// TIA Portal V20 program export: 1 tag tables, 54 data types, 39 data blocks, 33 code blocks (in call order from the OBs), 10 instance data blocks

VAR_GLOBAL   // PLC tag table "默认变量表"
   Clock_Byte AT %MB0 : Byte;
   Clock_10Hz AT %M0.0 : Bool;
   Clock_5Hz AT %M0.1 : Bool;
   "Clock_2.5Hz" AT %M0.2 : Bool;
   Clock_2Hz AT %M0.3 : Bool;
   "Clock_1.25Hz" AT %M0.4 : Bool;
   Clock_1Hz AT %M0.5 : Bool;
   "Clock_0.625Hz" AT %M0.6 : Bool;
   "Clock_0.5Hz" AT %M0.7 : Bool;
   System_Byte AT %MB1 : Byte;
   FirstScan AT %M1.0 : Bool;
   DiagStatusUpdate AT %M1.1 : Bool;
   AlwaysTRUE AT %M1.2 : Bool;
   AlwaysFALSE AT %M1.3 : Bool;
   PositioningAxis_1_Actor_Interface_AddressIn AT %I129.0 : "PD_TEL5_IN";
   PositioningAxis_1_Actor_Interface_AddressOut AT %Q132.0 : "PD_TEL5_OUT";
   滑台伺服S200_Actor_Interface_AddressIn AT %I260.0 : "PD_TEL105_IN";
   滑台伺服S200_Actor_Interface_AddressOut AT %Q260.0 : "PD_TEL105_OUT";
   RLO_1 AT %M100.0 : Bool;
   RLO_0 AT %M100.1 : Bool;
   FirstCycle AT %M100.2 : Bool;
   S120正限位 AT %I0.0 : Bool;
   s120负限位 AT %I0.1 : Bool;
   s120原点信号 AT %I0.2 : Bool;
   滑台伺服S200_Actor_Interface_TorqueDataAddressIn AT %I280.0 : "PD_TEL750_IN";
   滑台伺服S200_Actor_Interface_TorqueDataAddressOut AT %Q280.0 : "PD_TEL750_OUT";
   S200原点信号 AT %I0.3 : Bool;
   S200正限位 AT %I0.4 : Bool;
   S200负限位 AT %I0.5 : Bool;
   Tag_1 AT %M10.5 : Bool;
   Tag_2 AT %M10.6 : Bool;
END_VAR
VAR_GLOBAL CONSTANT   // user constants
   PN_DevDiag_MaxModules_UserConst : Int := 128;   // Maximale Anzahl der Module in einer ET-Station (z.B. ET200...); WICHTIG: um Zykluszeit und Speicherplatz zu optimieren mögl. kleinen Wert hier einstellen / Max number of modules, for optimization of scantime and memory space keep small / Max 数量 of modules, 给 optimization of scantime 和 内存 space keep small
   PN_DevDiag_MaxDevices_UserConst : Int := 255;   // Maximale Anzahl der PN-Devices; WICHTIG: um Zykluszeit und Speicherplatz zu optimieren mögl. kleinen Wert hier einstellen / Max number of PN-devices, for optimization of scantime and memory space keep small / Max 数量 of PN-devices, 给 optimization of scantime 和 内存 space keep small
   Type_HMI : Int := 101;   // SICAR HMI / HMI
   "Type_HMI+External" : Int := 102;   // SICAR HMI&Ext. / HMI&External / SICAR HMI&外部
   Type_External : Int := 103;   // SICAR Ext / External / SICAR 外部
   Type_OperatorPanel : Int := 105;   // SICAR OperatorPanel / OperatorPanel
   No_of_DataSets_Counter : Int := 8;   // Anzahl Datensätze Zähler / Number of data sets Counter / 数量 of 数据 sets 计数器
   No_of_DataSets_ShiftCounter : Int := 8;   // Anzahl Datensätze Schichtzähler / Number of data sets Shift Counter / 数量 of 数据 sets 工作轮班 计数器
   No_of_DataSets_CycleTimer : Int := 8;   // Anzahl Datensätze Taktzeiten / Number of data sets Cycle Timer / 数量 of 数据 sets 周期 记时器
   No_of_DataSets_LimitValues : Int := 8;   // Anzahl Datensätze Grenzwerte / Number of data sets Limit Value / 数量 of 数据 sets 限制 值
   No_Drives : Int := 2;   // Anzahl Antriebe / Number of drives / 数量 of 驱动
   No_UserOperation_screens : Int := 2;   // Anzahl Anwender Bedien-Bilder / Number of UserOperation screens / 数量 of UserOperation screens
   No_OperationMODE : Int := 5;   // Anzahl verwendeter Betriebsarten Breiche (max.: 12) / Number of used operation mode areas (max.: 12 ) / 数量 of used 运行 模式 areas (max.: 12 )
   No_HMI_PANEL : Int := 5;   // Anzahl verwendeter HMI/Panel (Max.: 40: 8 HMIs + 32 Panels) / Number of used HMI/Panel (Max.: 40: 8 HMIs + 32 Panels) / 数量 of used HMI/Panel (Max.: 40: 8 HMIs + 32 Panels)
   EQUIPMENTDATA_STEPHISTORYLENGTH : Int := 149;   // Equipment Data Step History Array Length / 设备 数据 步 历史 Array 长度
   EQUIPMENTDATA_ACTIVEALARMSLENGTH : Int := 9;   // Equipment Data Active Alarms Array Length / 设备 数据 现行 警报 Array 长度
   No_Reader : Int := 5;   // Anzahl Lesestellen / Number of reader / 数量 of 读码器
   No_Fixtures : Int := 2;
   No_Valves : Int := 4;
   No_PP : Int := 4;
   OpMode07_No_Robot : Int := 4;   // Anzahl Antriebe / Number of Robots
   No_ES : Int := 4;   // Anzahl Antriebe / Number of drives
   No_GS : Int := 1;   // Anzahl Antriebe / Number of drives
   No_LC : Int := 1;   // Anzahl Antriebe / Number of drives
   No_LS : Int := 1;   // Anzahl Antriebe / Number of drives
   Single_Input : Int := 1;
   OSSD_Input : Int := 5;
   OP_Sum : SInt := 2;   // 工位总数
   HMI_AXISCTRL_COUNT_AXES_UPPER_LIM : Int := 5;   // Upper limit for number of axes in HMI (maximum number - 1)
END_VAR

TYPE "ConvHMICMD"
   STRUCT
      StationOnly : Bool;   // Run Within Station Only
      SafetyTest : Bool;   // Safety Test
      Spare1 : Bool;   // Spare
      Spare2 : Bool;   // Spare
      Spare3 : Bool;   // Spare
      Spare4 : Bool;   // Spare
      Spare5 : Bool;   // Spare
      Spare6 : Bool;   // Spare
      Spare7 : Bool;   // Spare
      Spare8 : Bool;   // Spare
      Spare9 : Bool;   // Spare
      Spare10 : Bool;   // Spare
      Spare11 : Bool;   // Spare
      Spare12 : Bool;   // Spare
      Spare13 : Bool;   // Spare
      Spare14 : Bool;   // Spare
      Spare15 : Bool;   // Spare
      Spare16 : Bool;   // Spare
      Spare17 : Bool;   // Spare
      Spare18 : Bool;   // Spare
      Spare19 : Bool;   // Spare
      Spare20 : Bool;   // Spare
      Spare21 : Bool;   // Spare
      Spare22 : Bool;   // Spare
      Spare23 : Bool;   // Spare
      Spare24 : Bool;   // Spare
      Spare25 : Bool;   // Spare
      Spare26 : Bool;   // Spare
      Spare27 : Bool;   // Spare
      Spare28 : Bool;   // Spare
      Spare29 : Bool;   // Spare
      Spare30 : Bool;   // Spare
   END_STRUCT;
END_TYPE

TYPE "InPut"
   STRUCT
      TrfInSetBegin : Bool;   // Command in from Graph / Load Begin: condition to start transfer IN set
      TrfInSetIntlkOk : Bool;   // Transfer IN Interlock Set OK
      TrfInResIntlkOk : Bool;   // Transfer IN Interlock Reset OKt
      TrfOutSetBegin : Bool;   // Unload Begin: condition to start transfer OUT set
      TrfOutSetIntlkOk : Bool;   // Transfer Out Interlock Set Ok
      TrfOutResIntlkOk : Bool;   // Transfer OUT Interlock Reset Ok
      TrfOutResBegin : Bool;
   END_STRUCT;
END_TYPE

TYPE "OutPut"
   STRUCT
      Active : Bool;   // Roller is Active
      TrfInSetRdyRcv : Bool;   // Ready to Receive: Signal to previous object set
      TrfInSetArrived : Bool;   // Body Arrived: Signal to previous object Set
      TrfInSetActive : Bool;   // Transfer in set active
      TrfInSetFinished : Bool;   // Transfer in set finished
      TrfOutSetRdyDlv : Bool;   // Ready to Deliver: Signal to next object set
      TrfOutSetTM : Bool;   // Transfer: Signal to next object set
      TrfOutSetActive : Bool;   // Transfer out set active
      TrfOutSetFinished : Bool;   // Transfer out set finished
      TrfInResRdyRcv : Bool;   // Ready to Receive: Signal to previous object Reset
      TrfInResArrived : Bool;   // Body Arrived: Signal to previous object Reset
      TrfInResActive : Bool;   // Transfer in Reset active
      TrfInResFinished : Bool;   // Transfer in Reset finished
      TrfOutResRdyDlv : Bool;   // Ready to Deliver: Signal to next object Reset
      TrfOutResTM : Bool;   // Transfer: Signal to next object Reset
      TrfOutResActive : Bool;   // Transfer out Reset active
      TrfOutResFinished : Bool;   // Transfer out Reset finished
      BodyInPosition : Bool;   // Body In Position / Body in Position on roller
      NoSkid : Bool;   // No Skid
      LSpdSet : Bool;   // Lower Speed Set
      HSpdSet : Bool;   // Hight Speed Set
      SelectLower : Bool;   // Selext Lower Speed
   END_STRUCT;
END_TYPE

TYPE "RollBed"
   STRUCT
      HMI : "H_HMI";
      G120 { S7_SetPoint := 'True'} : "H_Roller2W2S-G120PN";
      Config { S7_SetPoint := 'True'} : "RollerConvConfig";
      InPut : "InPut";
      OutPut : "OutPut";
   END_STRUCT;
END_TYPE

TYPE "RollerConvConfig"
   STRUCT
      DeadEnd : Bool;   // Dead End Disable Positiong Fault
      TrspNoLowSpeed : Bool;   // Input 14
      StopDetSetUsed : Bool;   // Input 0
      LowSpeedDetSetUsed : Bool;   // Low Speed Det Used
      LowSpeedDetSetConstOn : Bool;   // Low Speed Sensor Constant on
      StopDetResUsed : Bool;   // Stop detection Reset used
      LowSpeedDetResUsed : Bool;   // Input 10
      LowSpeedDetResConstOn : Bool;   // Lowspeed stop detection Constant On
      TrainActivatedSet : Bool;   // Train transport used set direction
      TrfInSetUsed : Bool;   // Transfer In Set Used
      TrfOutSetUsed : Bool;   // Transfer Out Reset Used
      TrainActivatedRes : Bool;   // Train transport used Reset direction
      TrfInResUsed : Bool;   // Transfer In Reset Used
      TrfOutResUsed : Bool;   // Transfer Out Reset Used
      EnableAlarmHW : Bool := TRUE;   // Enable Alarm hardware (e.g. Safetyswitch, Motorprotector, detections)
      EnableAlarmTransfer : Bool;   // Enable Alarm transfer (e.g. Transfer in , transfer out)
      EnableG120Reset : Bool;   // Enable Driver Reset
      EnableCheckSpeedOK : Bool;   // Enable Speed checking on the G120 Driver
      EnableSetpoint : Bool;   // Enable setpoint
      EnableRFG : Bool;   // Follow setpoint
      NotQuickStop : Bool;   // QuickStop function; When FALSE the QuickStop of the G120 is Active
      NotImmediateStop : Bool;   // Immediate function; When FALSE the immediate stop of the G120 is Active
      EnableBeltControlSetDet : Bool;   // Config Belt Control
      EnableBeltControlResDet : Bool;   // Config Belt Control
      SLSUsed : Bool;   // Profisafe SLS Configuration Used
      SafetySwUsed : Bool;   // Input 12
      SafetySwNc : Bool;   // Input 15
      ReleaseBrakeUsed : Bool;   // Input 13
      RearDetUsed : Bool;   // Input 9
      RevSwUsed : Bool;   // Input 8
      MotorProtectionUsed : Bool;   // Motorprotection Used
      MotorProtectionNc : Bool;   // Motorprotection NC
      InitDirection : Bool;   // Input 6
      ForceManual : Bool;   // Configuration
      Spare1 : Bool;   // Spare
      Spare2 : Bool;   // Spare
      Spare3 : Bool;   // Spare
      TrfMaxTime : DInt;   // Max allowed transfertime (millisec)
      RPMSpeed : Real;   // Movment Rpm
      EnableRPMSpeed : Bool;   // Enable RPM Speed
      ReferenceSpeed : Int;   // Reference value for speed, stored in P2000 ot the SINAMICS
      ReferenceCurrent : Real;   // Reference value for current, stored in P2002 ot the SINAMICS
      ReferenceTorque : Real;   // Reference value for torque, stored in P2003 ot the SINAMICS
      DelaySetStopDet : Time := T#1ms;   // Delay Time Stop Detection
      DelayResStopDet : Time := T#1ms;   // Delay Time Stop Detection
      HWSubInput : HW_SUBMODULE;   // Address (input/output)
      HWSubOutput : HW_SUBMODULE;   // I/O
      SafetyAddress : HW_SUBMODULE;   // Address (input/output)
      FilterBeltControlSec : DInt;   // Filter In Seconds Belt Control
   END_STRUCT;
END_TYPE

TYPE "Rollerbed_Configuration"
   STRUCT
      StopDetSetUsed : Bool;
      LowSpeedDetSetUsed : Bool;
      LSpeedDetSetConstOn : Bool;
      TrainActivatedSet : Bool;
      TrfInSetUsed : Bool;
      TrfOutSetUsed : Bool;
      TrspNoLowSpeed : Bool;
      InitDirection : Bool;
      RevSwUsed : Bool;
      StopDetResUsed : Bool;
      LowSpeedDetResUsed : Bool;
      LSpeedDetResConstOn : Bool;
      TrainActivatedRes : Bool;
      TrfInResUsed : Bool;
      TrfOutResUsed : Bool;
      SafetySwNc : Bool;
      SafetySwUsed : Bool;
      ReleaseBrakeUsed : Bool;
      MotorProtectionSwNc : Bool;
      MotorProtectionUsed : Bool;
   END_STRUCT;
END_TYPE

TYPE "sPos16"
   STRUCT
      I_SS_bHome : Bool;   // 原点传感器
      I_SS_bFW : Bool := TRUE;   // 前限位
      I_SS_bBW : Bool := TRUE;   // 后限位
      I_CMD_bEnableAxis : Bool;   // 使能
      I_CMD_bResetAxis : Bool;   // 复位
      I_CMD_bjogForward : Bool;   // Taster Aufwärts / 正点
      I_CMD_bjogBackward : Bool;   // Taster Abwärts / 反点
      I_CMD_bmoveVelocity : Bool;   // 速度运行
      I_CMD_bstop : Bool;   // 停止
      I_CMD_bfastStop : Bool;   // 急停
      I_CMD_bHoming : Bool;   // 回零
      I_CMD_bGoToPos : Array[0..15] of Bool;   // Start Aufwärts in Automatik / 16个定位
      I_CMD_iGoToPos : Word;   // 16个定位 Word
      I_CMD_bCallAbsPos : Bool;   // 定位位置切换时，单独的定位按钮
      I_CMD_bRelPos : Bool;   // 相对定位
      I_CMD_MyBool : Array[0..5] of Bool;   // 临时变量
      I_Para_rJog_Speed : Array[0..2] of LReal;   // 点动速度/ACC/DEC/JERK
      I_Para_rMV_Speed : Array[0..2] of LReal;   // 速度运行速度/ACC/DEC/JERK
      I_Para_rStop_Dec : Array[0..1] of LReal;   // 速度运行速度/ACC/DEC/JERK
      I_Para_rEStop_Dec : Array[0..1] of LReal;   // 速度运行速度/ACC/DEC/JERK
      I_Para_iNum_Abspos : Int := 4;
      I_Para_rPos_Abs : Array[0..16] of LReal;   // 绝对定位目标位置
      I_Para_rSpeed_Abs : Array[0..16] of LReal;   // Endlage Unten / 绝对定位速度
      I_Para_rAcc_Set : Array[0..16] of LReal;   // 绝对定位加速度
      I_Para_rDec_Set : Array[0..16] of LReal;   // 绝对定位减速度
      I_Para_rJerk_Set : Array[0..16] of LReal;   // 绝对定位加加速度
      I_Para_rSpeedPercent : LReal := 20.0;   // Endlage Unten / 速度设定百分比
      I_Para_iHomeMode : Int;   // 回零方式
      I_Para_rHomePos : LReal;   // 回零位置
      O_Status_bAxisReady : Bool;   // 轴通讯正常
      O_Status_bAxisEnabled : Bool;   // 轴使能
      O_Status_bjogForward : Bool;   // 轴正点中
      O_Status_bjogBackward : Bool;   // 轴反点中
      O_Status_bHomed : Bool;   // 轴归零完成
      O_Status_bAtHome : Bool;   // 轴在零位
      O_Status_bSstill : Bool;   // 轴静止
      O_Status_bAxisBusy : Bool;   // 轴运行中
      O_Status_bAxisSyned : Bool;   // 同步上
      O_Status_bAxisError : Bool;   // 轴报警
      O_Status_bAtPos : Array[0..15] of Bool;   // Ausgang Aufwärts / 在目标位置上
      O_Status_bPosDone : Array[0..15] of Bool;   // 定位完成
      O_Status_bPosing : Array[0..15] of Bool;   // Ausgang Aufwärts / 定位中
      O_Status_bRelPosDone : Bool;   // 相对定位完成
      O_Status_rActPos : LReal;   // 实际位置
      O_Status_rActSpeed : LReal;   // 实际速度
      O_Status_iAxisFaultNum : UDInt;   // 轴报警代码
      O_Status_iDriveFaultNum : UDInt;   // 驱动报警代码
      O_Status_iFBStatus : Word;   // 运动功能块状态
      O_Status_iMCStatus : Word;   // 运动指令状态
      O_Status_rDriveTorque : LReal;   // 驱动扭矩
      O_Status_rDriveTemp : LReal;   // 驱动温度
      O_Status_rDriveRpm : LReal;   // 驱动转速
      O_Status_AxisName : WString[24] := WSTRING#'No axis';   // Name of axis
      O_Status_mybool : Array[0..5] of Bool;   // 备用
      O_Status_myLreal : Array[0..5] of LReal;   // 备用
      I_InLock_bEnableAxis : Bool;   // 使能
      I_InLock_bResetAxis : Bool;   // 复位
      I_InLock_bjogForward : Bool;   // Taster Aufwärts / 正点
      I_InLock_bjogBackward : Bool;   // Taster Abwärts / 反点
      I_InLock_bmoveVelocity : Bool;   // 速度运行
      I_InLock_bstop : Bool;   // 停止
      I_InLock_bfastStop : Bool;   // 急停
      I_InLock_bHoming : Bool;   // 回零
      I_InLock_bGoToPos : Array[0..16] of Bool;   // Start Aufwärts in Automatik / 16个定位
      I_InLock_iGoToPos : Word;   // 16个定位 Word
      I_InLock_bCallAbsPos : Bool;   // 定位位置切换时，单独的定位按钮
      I_InLock_bRelPos : Bool;   // 相对定位
      I_InLock_MyBool : Array[0..5] of Bool;   // 临时变量
      I_HMI_bEnableAxis : Bool;   // 使能
      I_HMI_bResetAxis : Bool;   // 复位
      I_HMI_bjogForward : Bool;   // Taster Aufwärts / 正点
      I_HMI_bjogBackward : Bool;   // Taster Abwärts / 反点
      I_HMI_bmoveVelocity : Bool;   // 速度运行
      I_HMI_bstop : Bool;   // 停止
      I_HMI_bfastStop : Bool;   // 急停
      I_HMI_bHoming : Bool;   // 回零
      I_HMI_bGoToPos : Array[0..16] of Bool;   // Start Aufwärts in Automatik / 16个定位
      I_HMI_iGoToPos : Word;   // 16个定位 Word
      I_HMI_bCallAbsPos : Bool;   // 定位位置切换时，单独的定位按钮
      I_HMI_bRelPos : Bool;   // 相对定位
      I_HMI_MyBool : Array[0..5] of Bool;   // 临时变量
   END_STRUCT;
   // I_Para_rJog_Speed[0] := 10.0;
   // I_Para_rJog_Speed[1..2] := 30.0;
   // I_Para_rMV_Speed[0] := 20.0;
   // I_Para_rMV_Speed[1..2] := 30.0;
   // I_Para_rStop_Dec[0] := 30.0;
   // I_Para_rStop_Dec[1] := 50.0;
   // I_Para_rEStop_Dec[0..1] := 50.0;
   // I_Para_rPos_Abs[1] := 10.0;
   // I_Para_rPos_Abs[2] := 20.0;
   // I_Para_rPos_Abs[3] := 30.0;
   // I_Para_rPos_Abs[4] := 40.0;
   // I_Para_rPos_Abs[5] := 50.0;
   // I_Para_rPos_Abs[6] := 60.0;
   // I_Para_rPos_Abs[7] := 70.0;
   // I_Para_rPos_Abs[8] := 80.0;
   // I_Para_rPos_Abs[9] := 90.0;
   // I_Para_rPos_Abs[10] := 100.0;
   // I_Para_rPos_Abs[11] := 110.0;
   // I_Para_rPos_Abs[12] := 120.0;
   // I_Para_rPos_Abs[13] := 130.0;
   // I_Para_rPos_Abs[14] := 140.0;
   // I_Para_rPos_Abs[15] := 150.0;
   // I_Para_rPos_Abs[16] := 160.0;
   // I_Para_rSpeed_Abs[0..16] := 20.0;
   // I_Para_rAcc_Set[0..16] := 50.0;
   // I_Para_rDec_Set[0..16] := 50.0;
   // I_Para_rJerk_Set[0..16] := 50.0;
END_TYPE

TYPE "SHIFTMODEL_LIST_UDT"
   STRUCT
      ShiftmodelList_Zero { ExternalAccessible := 'False'; ExternalVisible := 'False'; ExternalWritable := 'False'; S7_SetPoint := 'True'} : "SHIFTMODEL-TIMES_1DAY_UDT";   // Alle Zeitwerte (TOD) gleich 00:00:00 / All Time values (TOD) are 00:00:00
      ShiftmodelList_1 { ExternalAccessible := 'False'; ExternalVisible := 'False'; ExternalWritable := 'False'; S7_SetPoint := 'True'} : "SHIFTMODEL-TIMES_1DAY_UDT";   // Schichtmodel Liste 1 (1 Tag) / Shiftmodel list 1 (1 day)
      ShiftmodelList_2 { ExternalAccessible := 'False'; ExternalVisible := 'False'; ExternalWritable := 'False'; S7_SetPoint := 'True'} : "SHIFTMODEL-TIMES_1DAY_UDT";   // Schichtmodel Liste 2 (1 Tag) / Shiftmodel list 2 (1 day)
      ShiftmodelList_3 { ExternalAccessible := 'False'; ExternalVisible := 'False'; ExternalWritable := 'False'; S7_SetPoint := 'True'} : "SHIFTMODEL-TIMES_1DAY_UDT";   // Schichtmodel Liste 3 (1 Tag) / Shiftmodel list 3 (1 day)
      ShiftmodelList_4 { ExternalAccessible := 'False'; ExternalVisible := 'False'; ExternalWritable := 'False'; S7_SetPoint := 'True'} : "SHIFTMODEL-TIMES_1DAY_UDT";   // Schichtmodel Liste 4 (1 Tag) / Shiftmodel list 4 (1 day)
      ShiftmodelList_5 { ExternalAccessible := 'False'; ExternalVisible := 'False'; ExternalWritable := 'False'; S7_SetPoint := 'True'} : "SHIFTMODEL-TIMES_1DAY_UDT";   // Schichtmodel Liste 5 (1 Tag) / Shiftmodel list 5 (1 day)
      ShiftmodelList_6 { ExternalAccessible := 'False'; ExternalVisible := 'False'; ExternalWritable := 'False'; S7_SetPoint := 'True'} : "SHIFTMODEL-TIMES_1DAY_UDT";   // Schichtmodel Liste 6 (1 Tag) / Shiftmodel list 6 (1 day)
      ShiftmodelList_7 { ExternalAccessible := 'False'; ExternalVisible := 'False'; ExternalWritable := 'False'; S7_SetPoint := 'True'} : "SHIFTMODEL-TIMES_1DAY_UDT";   // Schichtmodel Liste 7 (1 Tag) / Shiftmodel list 7 (1 day)
      ShiftmodelList_8 { ExternalAccessible := 'False'; ExternalVisible := 'False'; ExternalWritable := 'False'; S7_SetPoint := 'True'} : "SHIFTMODEL-TIMES_1DAY_UDT";   // Schichtmodel Liste 8 (1 Tag) / Shiftmodel list 8 (1 day)
      ShiftmodelList_9 { ExternalAccessible := 'False'; ExternalVisible := 'False'; ExternalWritable := 'False'; S7_SetPoint := 'True'} : "SHIFTMODEL-TIMES_1DAY_UDT";   // Schichtmodel Liste 9 (1 Tag) / Shiftmodel list 9 (1 day)
      ShiftmodelList_10 { ExternalAccessible := 'False'; ExternalVisible := 'False'; ExternalWritable := 'False'; S7_SetPoint := 'True'} : "SHIFTMODEL-TIMES_1DAY_UDT";   // Schichtmodel Liste 10 (1 Tag) / Shiftmodel list 10 (1 day)
      Shiftmodel_WeekDay { ExternalAccessible := 'False'; ExternalVisible := 'False'; ExternalWritable := 'False'; S7_SetPoint := 'True'} : Array[1..7] of "SHIFTMODEL-TIMES_1DAY_UDT";   // Schichtmodel 1 Woche (1: Sunday, 2: Monday, 3: Thuesday, 4: Wednesday, 5: Thursday, 6: Friday, 7: Saturday) / Shiftmodel 1 week (1: Sunday, 2: Monday, 3: Thuesday, 4: Wednesday, 5: Thursday, 6: Friday, 7: Saturday)
   END_STRUCT;
END_TYPE

TYPE "RFID_BALLUFF_UDT"
   STRUCT
      Start : Bool;
      job_Type : Int;
      Adr_Recieve : Int;
      Adr_Send : Int;
      Addr_CodeTag : Int;
      Length_CodeTag : Int;
   END_STRUCT;
END_TYPE

TYPE "UDT_RFID_Basic_Data"
   STRUCT
      Pallet_ID : Int;   // 托盘号
      Repair_Status : Int;   // 返修标致（0：无状态，1：正常件，2：返修件）
      Reserves_1 : Int;   // 预留
      Reserves_2 : Int;   // 预留
      Reserves_3 : Int;   // 预留
      Reserves_4 : Int;   // 预留
      Reject_Stn_Number : String[8];   // 拒绝工位（由不合格工位写入）
      UpLoad_Stn_Number : String[8];   // 上线工位（返修上线工位写入）
      Reserves_5 : Int;   // 预留
      PLCProductWorkOrderID : String[66];   // 产品工单号数据
      PLCProductModelID : String[32];   // 产品型号信息
      PLCProductRecipeID : Word;   // 产品配方号数据
      PLCProductSN : String[96];   // 产品序列号
      PLCProductPN : String[96];   // 产品批次号
      PLCCurrentProductSN : String[96];   // 当前处理的产品序列号
      PLCProductCustomerSN : String[96];   // 产品客户序列号
      PLCProductCustomerSNType : Word;   // 产品客户序列号类型
      Reserves_6 : Int;   // 预留
      Reserves_7 : Int;   // 预留
      Reserves_8 : Int;   // 预留
      Reserves_9 : Int;   // 预留
   END_STRUCT;
END_TYPE

TYPE "UDT_RFID_STN_Data"
   STRUCT
      Station_Task : Byte;   // 工位建造状态（0:未完成 1:接受 2:拒绝）
      TASK_01 : Byte;   // 任务1状态（0:未完成 1:接受 2:拒绝）
      TASK_02 : Byte;   // 任务2状态（0:未完成 1:接受 2:拒绝）
      TASK_03 : Byte;   // 任务3状态（0:未完成 1:接受 2:拒绝）
      TASK_04 : Byte;   // 任务4状态（0:未完成 1:接受 2:拒绝）
      TASK_05 : Byte;   // 任务5状态（0:未完成 1:接受 2:拒绝）
      TASK_06 : Byte;   // 任务6状态（0:未完成 1:接受 2:拒绝）
      TASK_07 : Byte;   // 任务7状态（0:未完成 1:接受 2:拒绝）
      TASK_08 : Byte;   // 任务8状态（0:未完成 1:接受 2:拒绝）
      TASK_09 : Byte;   // 任务9状态（0:未完成 1:接受 2:拒绝）
   END_STRUCT;
END_TYPE

TYPE "VAR_RFID_UDT_BALLUFE"
   STRUCT
      Pallte_On { ExternalAccessible := 'False'; ExternalVisible := 'False'; ExternalWritable := 'False'} : Bool;
      Init { ExternalAccessible := 'False'; ExternalVisible := 'False'; ExternalWritable := 'False'} : Bool;   // 初始化
      Read_Req { ExternalAccessible := 'False'; ExternalVisible := 'False'; ExternalWritable := 'False'} : Bool;
      Write_Req { ExternalAccessible := 'False'; ExternalVisible := 'False'; ExternalWritable := 'False'} : Bool;
      Dyn { ExternalAccessible := 'False'; ExternalVisible := 'False'; ExternalWritable := 'False'} : Bool;   // 动态读写
      CT_Type { ExternalAccessible := 'False'; ExternalVisible := 'False'; ExternalWritable := 'False'} : Bool;   // 编码器类型
      IO_Start { ExternalAccessible := 'False'; ExternalVisible := 'False'; ExternalWritable := 'False'} : Int;
      IO_Length { ExternalAccessible := 'False'; ExternalVisible := 'False'; ExternalWritable := 'False'} : Int;
      CT_Length_R { ExternalAccessible := 'False'; ExternalVisible := 'False'; ExternalWritable := 'False'} : Int;
      CT_Length_W { ExternalAccessible := 'False'; ExternalVisible := 'False'; ExternalWritable := 'False'} : Int;
      Send_DB { ExternalAccessible := 'False'; ExternalVisible := 'False'; ExternalWritable := 'False'} : Int;
      Send_Adr { ExternalAccessible := 'False'; ExternalVisible := 'False'; ExternalWritable := 'False'} : Int;
      Recv_DB { ExternalAccessible := 'False'; ExternalVisible := 'False'; ExternalWritable := 'False'} : Int;
      Recv_Adr { ExternalAccessible := 'False'; ExternalVisible := 'False'; ExternalWritable := 'False'} : Int;
      Read_Finished { ExternalAccessible := 'False'; ExternalVisible := 'False'; ExternalWritable := 'False'} : Bool;
      Write_Finished { ExternalAccessible := 'False'; ExternalVisible := 'False'; ExternalWritable := 'False'} : Bool;
      Error { ExternalAccessible := 'False'; ExternalVisible := 'False'; ExternalWritable := 'False'} : Bool;
      ErrorNum { ExternalAccessible := 'False'; ExternalVisible := 'False'; ExternalWritable := 'False'} : Int;
      Dig_In { ExternalAccessible := 'False'; ExternalVisible := 'False'; ExternalWritable := 'False'} : Bool;
      CT_Present { ExternalAccessible := 'False'; ExternalVisible := 'False'; ExternalWritable := 'False'} : Bool;
   END_STRUCT;
END_TYPE

TYPE "MOTOR_LOCK_HMI_UDT"
   STRUCT
      State : DWord;   // Status Tec_Unit / State Tec_unit
      Plant_Identifier : WString[24];   // Betriebsmittel Kennzeichen / Plant identifier
      Move : Word;   // Schnittstelle Bewegungen / Interface Movement/Position
      Position : DWord;   // Schnittstelle Positionen 1-8 / Interface Position
      Alarm : Word;   // Störungen / Alarms
      State_Colour : SInt;   // Status Farbschema / State colour code
      HMI_Control_No : Int;   // HMI-Control Nummer / HMI-Control number
      OPModeArea { ExternalWritable := 'False'} : USInt;   // BA-Bereich / OPMode area
   END_STRUCT;
END_TYPE

TYPE "UDT_FIXTURE_IF"
   STRUCT
      Valves : Array[1..10] of "UDT_VALVE";
      PP : Array[1..35] of "PP_INTERFACE_UDT";
      Process_Complete : Array[1..16] of Bool;
      Work_Pos : Bool;
      Home_Pos : Bool;
      AtKnownPos : Bool;
   END_STRUCT;
END_TYPE

TYPE "UDT_VALVE"
TITLE = DEMO
// Autor: SICAR / Autor: Tesla
   STRUCT
      Auto_Work : Bool;   // Cmd To Move Valve To Work / Cmd 到 移动 汽阀 到 工作位
      Auto_Home : Bool;   // Cmd To Move Valve To Home / Cmd 到 移动 汽阀 到 原位
      At_Work : Bool;   // Status At Work / 状态 在 工作位
      At_Home : Bool;   // Status At Home / 状态 在 原位
      Enable_Work : Bool;   // interlock to move valve to Work / 互锁 到 移动 汽阀 到 工作位
      Enable_Home : Bool;   // interlock to move valve to Home / 互锁 到 移动 汽阀 到 原位
      General_Alarm : Bool;
      Known_Position : Bool;
      Position : "VALVE_POSITION_UDT";   // Feedback from Sensors / 反馈 从 Sensors
   END_STRUCT;
END_TYPE

TYPE "Udt_M200D_IN"
   STRUCT
      "Ready (automatic)" : Bool;
      "Motor on" : Bool;
      "Group fault" : Bool;
      "Group warning" : Bool;
      "Input 1_Stop" : Bool;
      "Input 2_Ocuupy" : Bool;
      "Input 3" : Bool;
      "Input 4" : Bool;
      "Current motor current Icurr % Bit 0" : Bool;
      "Current motor current Icurr % Bit 1" : Bool;
      "Current motor current Icurr % Bit 2" : Bool;
      "Current motor current Icurr % Bit 3" : Bool;
      "Current motor current Icurr % Bit 4" : Bool;
      "Current motor current Icurr % Bit 5" : Bool;
      "Manual mode local mode" : Bool;
      "Ramp operation" : Bool;
   END_STRUCT;
END_TYPE

TYPE "Udt_M200D_OUT"
   STRUCT
      "Motor CW" : Bool;
      "Motor CCW" : Bool;
      "Control for brake" : Bool;
      "Trip reset" : Bool;
      "Emergency start" : Bool;
      "Self-test" : Bool;
      Unassigned1 : Bool;
      Unassigned2 : Bool;
      "Output 1" : Bool;
      "Output 2" : Bool;
      Unassigned3 : Bool;
      Unassigned4 : Bool;
      Unassigned5 : Bool;
      Unassigned6 : Bool;
      Unassigned7 : Bool;
      "Disable quick stop" : Bool;
   END_STRUCT;
END_TYPE

TYPE "PLC_STATUS_UDT"
   STRUCT
      RUN_STOP : Int;   // RUN/STOP LED (Yellow/Green) / 运行/停止 LED (黄/Green)
      ER_ERROR : Int;   // ERROR LED (Red) / 错误 LED (红)
      MT_MAINT : Int;   // MAINT LED (Yellow) / MAINT LED (黄)
      QSTATUS : Bool;   // FAIL SAFE STATUS / 安全失败 状态
      RIOforFA_VALUE_STATUS : Bool;   // FAIL SAFE STATUS / 安全失败 状态
      F_DEVICE_PASSIVATED : Bool;   // FAIL SAFE STATUS / 安全失败 状态
   END_STRUCT;
END_TYPE

TYPE "HMIAxisCtrl_typeInterface"
TITLE = HMIAxisCtrl_typeInterface
// Support: tech.team.motioncontrol@siemens.com 
// Fax: +49 (0) 9131/98-1297
   STRUCT
      actualValues { S7_SetPoint := 'True'} : "HMIAxisCtrl_typeActualValues";   // Actual values of axis
      general { S7_SetPoint := 'True'} : "HMIAxisCtrl_typeGeneral";   // General axis information
      internal { S7_SetPoint := 'True'} : "HMIAxisCtrl_typeInternal";   // Internal variable for visualization
      inputs { S7_SetPoint := 'True'} : "HMIAxisCtrl_typeInputs";   // Inputs AxisCtrl
      outputs { S7_SetPoint := 'True'} : "HMIAxisCtrl_typeOutputs";   // Outputs AxisCtrl
      configuration { S7_SetPoint := 'True'} : "LAxisCtrl_typeAxisConfig";   // Config AxisCtrl
      diagnostics { S7_SetPoint := 'True'} : "LAxisCtrl_typeDiagnostics";   // Diagnostics AxisCtrl
   END_STRUCT;
   // general.axisType := 0;
END_TYPE

TYPE "sAxis"
   STRUCT
      I_SS { S7_SetPoint := 'True'} : "sAxis_SS";
      I_CMD { S7_SetPoint := 'True'} : "sAxis_CMD";
      I_Para { S7_SetPoint := 'True'} : "sAxis_Para";
      O_Status { S7_SetPoint := 'True'} : "sAxis_Status";
      I_InLock { S7_SetPoint := 'True'} : "sAxis_InLock";
      I_HMI { S7_SetPoint := 'True'} : "sAxis_HMI";
   END_STRUCT;
END_TYPE

TYPE "sAxis_CMD"
   STRUCT
      bEnableAxis : Bool;   // 使能
      bResetAxis : Bool;   // 复位
      bjogForward : Bool;   // Taster Aufwärts / 正点
      bjogBackward : Bool;   // Taster Abwärts / 反点
      bmoveVelocity : Bool;   // 速度运行
      bstop : Bool;   // 停止
      bfastStop : Bool;   // 急停
      bHoming : Bool;   // 回零
      bGoToPos : Array[0..16] of Bool;   // Start Aufwärts in Automatik / 16个定位
      iGoToPos : Word;   // 16个定位 Word
      bCallAbsPos : Bool;   // 定位位置切换时，单独的定位按钮
      bRelPos : Bool;   // 相对定位
      MyBool : Array[0..5] of Bool;   // 临时变量
   END_STRUCT;
END_TYPE

TYPE "sAxis_HMI"
   STRUCT
      bEnableAxis : Bool;   // 使能
      bjogForward : Bool;   // Taster Aufwärts / 正点
      bjogBackward : Bool;   // Taster Abwärts / 反点
      bmoveVelocity : Bool;   // 速度运行
      bstop : Bool;   // 停止
      bHoming : Bool;   // 回零
      bGoToPos : Array[0..16] of Bool;   // Start Aufwärts in Automatik / 16个定位
      iGoToPos : Word;   // 16个定位 Word
      bCallAbsPos : Bool;   // 定位位置切换时，单独的定位按钮
      bRelPos : Bool;   // 相对定位
      MyBool : Array[0..5] of Bool;   // 临时变量
   END_STRUCT;
END_TYPE

TYPE "sAxis_InLock"
   STRUCT
      bEnableAxis : Bool;   // 使能
      bResetAxis : Bool;   // 复位
      bjogForward : Bool;   // Taster Aufwärts / 正点
      bjogBackward : Bool;   // Taster Abwärts / 反点
      bmoveVelocity : Bool;   // 速度运行
      bstop : Bool;   // 停止
      bfastStop : Bool;   // 急停
      bHoming : Bool;   // 回零
      bGoToPos : Array[0..16] of Bool;   // Start Aufwärts in Automatik / 16个定位
      iGoToPos : Word;   // 16个定位 Word
      bCallAbsPos : Bool;   // 定位位置切换时，单独的定位按钮
      bRelPos : Bool;   // 相对定位
      MyBool : Array[0..5] of Bool;   // 临时变量
   END_STRUCT;
END_TYPE

TYPE "sAxis_Para"
   STRUCT
      rJog_Speed : Array[0..2] of LReal;   // 点动速度/ACC/DEC/JERK
      rMV_Speed : Array[0..2] of LReal;   // 速度运行速度/ACC/DEC/JERK
      rStop_Dec : Array[0..1] of LReal;
      rEStop_Dec : Array[0..1] of LReal;
      iNum_Abspos : Int := 4;
      rPos_Abs : Array[0..16] of LReal;   // 绝对定位目标位置 / Over travel switch set
      rSpeed_Abs : Array[0..16] of LReal;   // Endlage Unten / 绝对定位速度
      rAcc_Set : Array[0..16] of LReal;   // 绝对定位加速度 / Overtravel switch Reset
      rDec_Set : Array[0..16] of LReal;   // 绝对定位减速度 / Belt check sensor
      rJerk_Set : Array[0..16] of LReal;   // 绝对定位加加速度
      rSpeedPercent : LReal := 20.0;   // Endlage Unten / 速度设定百分比
      iHomeMode : Int;   // 回零方式
      rHomePos : LReal;   // 回零位置
   END_STRUCT;
   // rJog_Speed[0] := 10.0;
   // rJog_Speed[1..2] := 30.0;
   // rMV_Speed[0] := 20.0;
   // rMV_Speed[1..2] := 30.0;
   // rStop_Dec[0] := 30.0;
   // rStop_Dec[1] := 50.0;
   // rEStop_Dec[0..1] := 50.0;
   // rPos_Abs[1] := 10.0;
   // rPos_Abs[2] := 20.0;
   // rPos_Abs[3] := 30.0;
   // rPos_Abs[4] := 40.0;
   // rPos_Abs[5] := 50.0;
   // rPos_Abs[6] := 60.0;
   // rPos_Abs[7] := 70.0;
   // rPos_Abs[8] := 80.0;
   // rPos_Abs[9] := 90.0;
   // rPos_Abs[10] := 100.0;
   // rPos_Abs[11] := 110.0;
   // rPos_Abs[12] := 120.0;
   // rPos_Abs[13] := 130.0;
   // rPos_Abs[14] := 140.0;
   // rPos_Abs[15] := 150.0;
   // rPos_Abs[16] := 160.0;
   // rSpeed_Abs[0..16] := 20.0;
   // rAcc_Set[0..16] := 50.0;
   // rDec_Set[0..16] := 50.0;
   // rJerk_Set[0..16] := 50.0;
END_TYPE

TYPE "sAxis_SS"
   STRUCT
      bHome : Bool;   // 原点传感器
      bFW : Bool := TRUE;   // 前限位
      bBW : Bool := TRUE;   // 后限位
   END_STRUCT;
END_TYPE

TYPE "sAxis_Status"
   STRUCT
      bAxisReady : Bool;   // 轴通讯正常
      bAxisEnabled : Bool;   // 轴使能
      bjogForward : Bool;   // 轴正点中
      bjogBackward : Bool;   // 轴反点中
      bHomed : Bool;   // 轴归零完成
      bAtHome : Bool;   // 轴在零位
      bSstill : Bool;   // 轴静止
      bAxisBusy : Bool;   // 轴运行中
      bAxisSyned : Bool;   // 同步上
      bAxisError : Bool;   // 轴报警
      bAtPos : Array[0..15] of Bool;   // Ausgang Aufwärts / 在目标位置上
      bPosDone : Array[0..15] of Bool;   // 定位完成
      bPosing : Array[0..15] of Bool;   // Ausgang Aufwärts / 定位中
      bRelPosDone : Bool;   // 相对定位完成
      rActPos : LReal;   // 实际位置
      rActSpeed : LReal;   // 实际速度
      iAxisFaultNum : UDInt;   // 轴报警代码
      iDriveFaultNum : UDInt;   // 驱动报警代码
      iFBStatus : Word;   // 运动功能块状态
      iMCStatus : Word;   // 运动指令状态
      rDriveTorque : LReal;   // 驱动扭矩
      rDriveTemp : LReal;   // 驱动温度
      rDriveRpm : LReal;   // 驱动转速
      wAxisName : WString[24] := WSTRING#'No axis';   // Name of axis
      mybool : Array[0..5] of Bool;   // 备用
      myLreal : Array[0..5] of LReal;   // 备用
   END_STRUCT;
END_TYPE

TYPE "udt_Andon"
   STRUCT
      inpResetReq : Bool;
      inpPressFixedStop : Bool;
      inpPressTempStop { ExternalAccessible := 'False'; ExternalVisible := 'False'; ExternalWritable := 'False'} : Bool;
      inpTAE_StopRequestReset : Bool;
      inpTAE_FixedStop : Bool;
      inpTAE_TempStop : Bool;
      inpTAE_EOT_Reached : Bool;
      outFixedStop { ExternalAccessible := 'False'; ExternalVisible := 'False'; ExternalWritable := 'False'} : Bool;   // HW interface to the physical press button lamp / HW 接口 到 physical press 按钮 lamp
      outTempStop { ExternalAccessible := 'False'; ExternalVisible := 'False'; ExternalWritable := 'False'} : Bool;   // HW interface to the physical press button lamp / HW 接口 到 physical press 按钮 lamp
      Status : Int;
   END_STRUCT;
END_TYPE

TYPE "udt_BAE00TM"
   STRUCT
      PSU_Status : Bool;   // Power Supply On/Off / 电源 开/关
      Output_Drop : Bool;   // Output Drop (BDC3) / 输出 放下 (BDC3)
      Over_Temperature : Bool;   // Over Temperature (BDC2) / Over 温度 (BDC2)
      Over_Voltage : Bool;   // Over Voltage (BDC1) / Over 电压 (BDC1)
      Overload : Bool;   // Overload (BDC0) / 过载 (BDC0)
      Error_Code : Int;   // Error Code / 错误 Code
      Output_Voltage : Real;   // Output Voltage / 输出 电压
      Output_Current : Real;   // Output Current / 输出 电流
   END_STRUCT;
END_TYPE

TYPE "udt_BNI005H"
   STRUCT
      Output_Pin4_Control : Int;
      Output_Pin2_Control : Int;
      Restart_Pin4_Control : Int;
      Restart_Pin2_Control : Int;
      IOL_Diagnosis_Enable : Int;
      Inputs_Pin4 : Byte;
      Inputs_Pin2 : Byte;
      Actuator_Shutdown_Pin4 : Byte;
      Actuator_Shotdown_Pin2 : Byte;
      Actuator_Warning_Pin4 : Byte;
      Actuator_Warning_Pin2 : Byte;
      Sensor_Supply_Short_Circuit : Byte;
      IOL_Comm_Status : Byte;
   END_STRUCT;
END_TYPE

TYPE "udt_Manual_Station"
   STRUCT
      Config : Struct
         TaktTime : Time;
         OperatorTaskTime : Time;
         FlowStepName : WString[10];
         NextStationFlowStepName : WString[10];
         StationNumber : Int;
         StationName : String[6];
         StationBypass : Bool;
         TAE_Enable : Bool;
         BlockedTimerPreset : Time;
      END_STRUCT;
      Takt : Struct
         RunTimer : Bool;
         ResetTimer : Bool;
         TimerPreset : Time;
         TimerValue : Time;
      END_STRUCT;
      OPMode : "OPMODE_OUT_UDT";
   END_STRUCT;
END_TYPE

TYPE "IDENT_IF_UDT"
   STRUCT
      ENABLE_MAN_CTRL { ExternalAccessible := 'False'; ExternalVisible := 'False'; ExternalWritable := 'False'} : Bool;
      ENABLE_WRITE_TAG_ID { ExternalAccessible := 'False'; ExternalVisible := 'False'; ExternalWritable := 'False'} : Bool;
      CMD_INIT { ExternalAccessible := 'False'; ExternalVisible := 'False'; ExternalWritable := 'False'} : Bool;
      CMD_READ { ExternalAccessible := 'False'; ExternalVisible := 'False'; ExternalWritable := 'False'} : Bool;
      CMD_WRITE { ExternalAccessible := 'False'; ExternalVisible := 'False'; ExternalWritable := 'False'} : Bool;
      RESET { ExternalAccessible := 'False'; ExternalVisible := 'False'; ExternalWritable := 'False'} : Bool;
      ALARM { ExternalAccessible := 'False'; ExternalVisible := 'False'; ExternalWritable := 'False'} : Bool;
      WARNING { ExternalAccessible := 'False'; ExternalVisible := 'False'; ExternalWritable := 'False'} : Bool;
      INIT_DONE { ExternalAccessible := 'False'; ExternalVisible := 'False'; ExternalWritable := 'False'} : Bool;
      READ_DONE { ExternalAccessible := 'False'; ExternalVisible := 'False'; ExternalWritable := 'False'} : Bool;
      WRITE_DONE { ExternalAccessible := 'False'; ExternalVisible := 'False'; ExternalWritable := 'False'} : Bool;
      WRITE_DATA_OK { ExternalAccessible := 'False'; ExternalVisible := 'False'; ExternalWritable := 'False'} : Bool;
      INIT_ERROR { ExternalAccessible := 'False'; ExternalVisible := 'False'; ExternalWritable := 'False'} : Bool;
      READ_ERROR { ExternalAccessible := 'False'; ExternalVisible := 'False'; ExternalWritable := 'False'} : Bool;
      WRITE_ERROR { ExternalAccessible := 'False'; ExternalVisible := 'False'; ExternalWritable := 'False'} : Bool;
      TAG_PRESENCE { ExternalAccessible := 'False'; ExternalVisible := 'False'; ExternalWritable := 'False'} : Bool;
   END_STRUCT;
END_TYPE

TYPE "Udt_CarCode"
   STRUCT
      Plant_Identifier : WString[24];
      CarCode : Int;   // BadyCode
      Reserve1 : Int;
      Reserve2 : Int;
      Reserve3 : Int;
      Reserve4 : Int;
   END_STRUCT;
END_TYPE

TYPE "HMIAxisCtrl_typeActualValues"
TITLE = HMIAxisCtrl_typeActualValues
// Support: tech.team.motioncontrol@siemens.com 
// Fax: +49 (0) 9131/98-1297
   STRUCT
      actualVelocity : LReal;   // Actual value of velocity
      actualPosition : LReal;   // Actual value of position
      targetPosition : LReal;   // Actual value of target position
      isHomed : Bool;   // TRUE: Axis is homed
      brakeIsOpen : Bool;   // TRUE: Brake is open
      axisAlarm : UDInt;   // Number of the technology alarm
      axisError : Bool;   // TRUE: Axis has error
      errorDetailReaction : DInt;   // Effective alarm reaction
   END_STRUCT;
END_TYPE

TYPE "HMIAxisCtrl_typeGeneral"
TITLE = HMIAxisCtrl_typeGeneral
// Support: tech.team.motioncontrol@siemens.com 
// Fax: +49 (0) 9131/98-1297
   STRUCT
      axisType : DInt := 0;   // 1:SpeedAxis; 2:PosSyncAxis; 3:ExternalEncoder
      axisName : WString[24] := WSTRING#'No axis';   // Name of axis
      lengthUnit : UDInt;   // Unit for position
      velocityUnit : UDInt;   // Unit for velocity
      torqueForceUnit : UDInt;   // Unit for torque/Unit for force
      motionType : DInt := -1;   // Indication of axis or motion type: 0: Linear axis or motion 1: Rotary axis or motion
      encoderType : Int := 0;   // 1: Axis with incremental encoder; 2: Incremental external encoder; 3: Absolute external encoder or axis with absolute encoder
      moduloActive : Bool;   // TRUE: modulo active
      moduloLength : LReal;   // Modulo length
      limitBase : DInt := -1;   // Torque limiting. 0: Motor side; 1: Load side
      brakeExistent : Bool;   // TRUE: Brake existent
   END_STRUCT;
END_TYPE

TYPE "HMIAxisCtrl_typeInputs"
TITLE = HMIAxisCtrl_typeInputs
// Support: tech.team.motioncontrol@siemens.com 
// Fax: +49 (0) 9131/98-1297
   STRUCT
      enable : Bool;   // TRUE: Enable functionality of FB
      enableAxis : Bool;   // TRUE: Set axis enable; FALSE: Remove axis enable
      resetAxis : Bool;   // Rising edge: Acknowledgement of technology alarms or restart of the axis (depending on configuration)
      jogForward : Bool;   // Rising edge: Move an axis in jog mode (forward); Falling edge: Stop jogging
      jogBackward : Bool;   // Rising edge: Move an axis in jog mode (backward); Falling edge: Stop jogging
      moveVelocity : Bool;   // Rising edge: Move an axis at constant velocity/speed
      stop : Bool;   // Rising edge: Brake an axis until it comes to a standstill
      fastStop : Bool;   // Rising edge: Brake an axis until it comes to a standstill (with fastStop dynamics)
      torqueLimiting : Bool;   // TRUE: Enable force/torque limiting
      homing : Bool;   // Rising edge: Home axis
      posRelative : Bool;   // Rising edge: Move an axis relative to its position when execution of the job began
      posAbsolute : Bool;   // Rising edge: Move an axis to an absolute position
      posSuperimposed : Bool;   // Rising edge: Start a superimposed positioning
      gearInRelative : Bool;   // Rising edge: Start a gearing operation (relative)
      gearInAbsolute : Bool;   // Rising edge: Start a gearing operation (absolute)
      camIn : Bool;   // Rising edge: Start a camming operation
      phasing : Bool;   // Rising edge: Start a phasing operation
      openBrake : Bool;   // TRUE: Open holding brake
   END_STRUCT;
END_TYPE

TYPE "HMIAxisCtrl_typeInternal"
TITLE = HMIAxisCtrl_typeInternal
// Support: tech.team.motioncontrol@siemens.com 
// Fax: +49 (0) 9131/98-1297
   STRUCT
      mode : Int := -1;   // Internal mode identifier; 1: Jog ; 2: Move; 3: Pos; 4: Homing; 5: Brake
      absoluteSelected : Bool;   // TRUE: Absolute positioning; FALSE: Relative positioning
      isPosRelative : Bool;   // TRUE: Show controls related to relative positioning
      isPosAbsoluteWithModulo : Bool;   // TRUE: Show controls related to absolute positioning (with modulo)
      isPosAbsoluteWithoutModulo : Bool;   // TRUE: Show controls related to absolute positioning (without modulo)
      isAxisWithIncrementalEncoder : Bool;   // TRUE: Show controls related to axis with incremental encoder
      isAxisWithAbsoluteEncoder : Bool;   // TRUE: Show controls related to axis with absolute encoder
      isNotExternalEncoder : Bool;   // TRUE: Show controls related to homing functionality of axis (not external encoder)
      velocity : LReal := -1.0;   // Internal variable for velocity input
      position : LReal := 0.0;   // Internal variable for position input
      acceleration : LReal := -1.0;   // Internal variable for acceleration input
      deceleration : LReal := -1.0;   // Internal variable for deceleration input
      jerk : LReal := -1.0;   // Internal variable for jerk input
   END_STRUCT;
END_TYPE

TYPE "HMIAxisCtrl_typeOutputs"
TITLE = HMIAxisCtrl_typeOutputs
// Support: tech.team.motioncontrol@siemens.com 
// Fax: +49 (0) 9131/98-1297
   STRUCT
      valid : Bool;   // TRUE: Valid set of outputs available at the FB
      busy : Bool;   // TRUE: FB is working and new output values can be expected
      error : Bool;   // TRUE: An error occurred while processing the FB
      status : Word;   // Current status of FB
      axisEnabled : Bool;   // TRUE: The technology object is enabled. Motion commands can be executed.
      resetActive : Bool;   // TRUE: Reset/Restart of the axis is active
      commandBusy : Bool;   // TRUE: The selected basic motion command is being executed
      commandDone : Bool;   // TRUE: The selected basic motion command has completed without error
      commandAborted : Bool;   // TRUE: The selected basic motion command has been aborted
      inVelocity : Bool;   // TRUE: The setpoint velocity/speed was reached and will be maintained
      inLimitation : Bool;   // TRUE: The drive is operating at the force/torque limit
      homingCommandBusy : Bool;   // TRUE: Homing command is being executed
      homingCommandDone : Bool;   // TRUE: Homing command has completed without error
      homingCommandAborted : Bool;   // TRUE: Homing command has been aborted
      superimposedBusy : Bool;   // TRUE: The selected superimposed motion command is being executed
      superimposedDone : Bool;   // TRUE: The selected superimposed motion command has completed without error
      superimposedAborted : Bool;   // TRUE: The selected superimposed motion command has been aborted
      inClamping : Bool;   // TRUE: The drive is kept at the fixed stop (clamping), the axis position is within the positioning tolerance
      startSync : Bool;   // TRUE: The axis is synchronizing to the leading axis
      inSync : Bool;   // TRUE: The axis is synchronized to the leading axis
      inSimulation : Bool;   // TRUE: Synchronous operation is being simulated
      jogSelected : Bool;   // TRUE: Jogging is active
      moveVelocitySelected : Bool;   // TRUE: Moving with constant velocity/speed is active
      stopSelected : Bool;   // TRUE: Stopping is active
      fastStopSelected : Bool;   // TRUE: Stopping is active (with fastStop dynamics)
      torqueLimitingSelected : Bool;   // TRUE: Force/Torque limiting is active
      homingSelected : Bool;   // TRUE: Homing is active
      posRelativeSelected : Bool;   // TRUE: Relative positioning is active
      posAbsoluteSelected : Bool;   // TRUE: Absolute positioning is active
      posSuperimposedSelected : Bool;   // TRUE: Superimposed positioning is active
      gearInRelativeSelected : Bool;   // TRUE: Relative gearing is active
      gearInAbsoluteSelected : Bool;   // TRUE: Absolute gearing is active
      camInSelected : Bool;   // TRUE: Camming is active
      phasingSelected : Bool;   // TRUE: Phasing is active
   END_STRUCT;
END_TYPE

TYPE "LAxisCtrl_typeAxisConfig"
TITLE = LAxisCtrl_typeAxisConfig
// Support: tech.team.motioncontrol@siemens.com 
// Fax: +49 (0) 9131/98-1297
   STRUCT
      generalSettings { S7_SetPoint := 'True'} : "LAxisCtrl_typeGeneralSettings";   // Configuration of general settings
      power { S7_SetPoint := 'True'} : "LAxisCtrl_typePower";   // Configuration of MC_POWER function
      jog { S7_SetPoint := 'True'} : "LAxisCtrl_typeJog";   // Configuration of JOG function
      moveVelocity { S7_SetPoint := 'True'} : "LAxisCtrl_typeMoveVelocity";   // Configuration of MC_MOVEVELOCITY function
      stop { S7_SetPoint := 'True'} : "LAxisCtrl_typeStop";   // Configuration of MC_HALT function
      fastStop { S7_SetPoint := 'True'} : "LAxisCtrl_typeFastStop";   // Configuration of MC_HALT function (alternative dynamics)
      torqueLimiting { S7_SetPoint := 'True'} : "LAxisCtrl_typeTorqueLimiting";   // Configuration of MC_TORQUELIMITING function
      homing { S7_SetPoint := 'True'} : "LAxisCtrl_typeHoming";   // Configuration of HOMING function
      posRelative { S7_SetPoint := 'True'} : "LAxisCtrl_typePosRelative";   // Configuration of MC_MOVERELATIVE function
      posAbsolute { S7_SetPoint := 'True'} : "LAxisCtrl_typePosAbsolute";   // Configuration of MC_MOVEABSOLUTE function
      posSuperimposed { S7_SetPoint := 'True'} : "LAxisCtrl_typePosSuperimposed";   // Configuration of MC_MOVESUPERIMPOSED function
      gearInRelative { S7_SetPoint := 'True'} : "LAxisCtrl_typeGearInRelative";   // Configuration of MC_GEARIN function
      gearInAbsolute { S7_SetPoint := 'True'} : "LAxisCtrl_typeGearInAbsolute";   // Configuration of MC_GEARIN_POS function
      camIn { S7_SetPoint := 'True'} : "LAxisCtrl_typeCamIn";   // Configuration of MC_CAMIN function
      phasing { S7_SetPoint := 'True'} : "LAxisCtrl_typePhasing";   // Configuration of MC_PHASING function
   END_STRUCT;
END_TYPE

TYPE "LAxisCtrl_typeDiagnostics"
TITLE = LAxisCtrl_typeDiagnostics
// Support: tech.team.motioncontrol@siemens.com 
// Fax: +49 (0) 9131/98-1297
   STRUCT
      status : Word := 16#0000;   // Status of FB when error occurred
      subfunctionStatus : Word := 16#0000;   // ErrorID of called subfunction
      basicMotionState : DInt := 0;   // Current basic motion state when error occurred
      superimposedMotionState : DInt := 0;   // Current superimposed motion state when error occurred
   END_STRUCT;
END_TYPE

TYPE "LAxisCtrl_typeCamIn"
TITLE = LAxisCtrl_typeCamIn
// Support: tech.team.motioncontrol@siemens.com 
// Fax: +49 (0) 9131/98-1297
   STRUCT
      masterOffset : LReal := 0.0;   // Offset of leading values of cam
      slaveOffset : LReal := 0.0;   // Offset of following values of cam
      masterScaling : LReal := 1.0;   // Scaling the leading values of the cam
      slaveScaling : LReal := 1.0;   // Scaling the following values of the cam
      masterSyncPosition : LReal := 0.0;   // Starting point in the cam/distance from the cam start with reference to the scaled cam
      syncProfileReference : DInt := 1;   // Synchronization profile (0: Synchronization using dynamic parameters; 1: Synchronization using leading value distance; 2: Direct synchronous setting)
      masterStartDistance : LReal := 0.0;   // Leading value distance (when "SyncProfileReference" = 1)
      velocity : LReal := -1.0;   // Velocity for synchronization (when "SyncProfileReference" = 0; Value > 0.0: The specified value is used; Value = 0.0: Not permitted; Value < 0.0: Use of the default value configured in the technology object)
      acceleration : LReal := -1.0;   // Acceleration for synchronization (when "SyncProfileReference" = 0; Value > 0.0: The specified value is used; Value = 0.0: Not permitted; Value < 0.0: Use of the default value configured in the technology object)
      deceleration : LReal := -1.0;   // Deceleration for synchronization (when "SyncProfileReference" = 0; Value > 0.0: The specified value is used; Value = 0.0: Not permitted; Value < 0.0: Use of the default value configured in the technology object)
      jerk : LReal := -1.0;   // Jerk for synchronization (when "SyncProfileReference" = 0; Value > 0.0: Smooth velocity profile, the specified value is used; Value = 0.0: Trapezoid velocity profile; Value < 0.0: Use of the default value configured in the technology object)
      applicationMode : DInt := 0;   // Application of the cam (0: Once/not cyclic; 1: Cyclic ; 2: Cyclic appending)
      syncDirection : DInt := 1;   // Direction for synchronization only in effect for axes with activated modulo setting (1: Forward direction; 2: Backward direction; 3: Shortest way)
   END_STRUCT;
END_TYPE

TYPE "LAxisCtrl_typeFastStop"
TITLE = LAxisCtrl_typeFastStop
// Support: tech.team.motioncontrol@siemens.com 
// Fax: +49 (0) 9131/98-1297
   STRUCT
      deceleration : LReal := -1.0;   // Deceleration for fast stop (Value > 0.0: The specified value is used; Value <= 0.0: emergency deceleration of the technology object is used)
      jerk : LReal := -1.0;   // Jerk for fast stop (Value > 0.0: Smooth velocity profile, the specified value is used; Value = 0.0: Trapezoid velocity profile; Value < 0.0: Use of the default value configured in the technology object)
      abortAcceleration : Bool := FALSE;   // TRUE: The acceleration is set to 0.0 at the start of the job, and the deceleration immediately builds up; FALSE: The current acceleration at the start of the job is reduced using the configured jerk. Afterwards, the deceleration builds up
      replaceStopPossible : Bool := FALSE;   // TRUE: Fast stop command can be replaced by another command
   END_STRUCT;
END_TYPE

TYPE "LAxisCtrl_typeGearInAbsolute"
TITLE = LAxisCtrl_typeGearInAbsolute
// Support: tech.team.motioncontrol@siemens.com 
// Fax: +49 (0) 9131/98-1297
   STRUCT
      ratioNumerator : DInt := 1;   // Gear ratio numerator
      ratioDenominator : DInt := 1;   // Gear ratio denominator
      masterSyncPosition : LReal := 0.0;   // Synchronous position of leading axis
      slaveSyncPosition : LReal := 0.0;   // Synchronous position of following axis
      syncProfileReference : DInt := 1;   // Type of synchronization (0: Synchronization using dynamic parameters; 1: Synchronization using leading value distance)
      masterStartDistance : LReal := 0.0;   // Leading value distance (when "SyncProfileReference" = 1)
      velocity : LReal := -1.0;   // Velocity for synchronization (when "SyncProfileReference" = 0; Value > 0.0: The specified value is used; Value = 0.0: Not permitted; Value < 0.0: Use of the default value configured in the technology object)
      acceleration : LReal := -1.0;   // Acceleration for synchronization (when "SyncProfileReference" = 0; Value > 0.0: The specified value is used; Value = 0.0: Not permitted; Value < 0.0: Use of the default value configured in the technology object)
      deceleration : LReal := -1.0;   // Deceleration for synchronization (when "SyncProfileReference" = 0; Value > 0.0: The specified value is used; Value = 0.0: Not permitted; Value < 0.0: Use of the default value configured in the technology object)
      jerk : LReal := -1.0;   // Jerk for synchronization (when "SyncProfileReference" = 0; Value > 0.0: Smooth velocity profile, the specified value is used; Value = 0.0: Trapezoid velocity profile; Value < 0.0: Use of the default value configured in the technology object)
      syncDirection : DInt := 1;   // Direction for synchronization only in effect for axes with activated modulo setting (1: Forward direction; 2: Backward direction; 3: Shortest way)
      ratioChangeOnTheFly : Bool := FALSE;   // TRUE: Changing gear ratio on-the-fly; FALSE: Ratio change requires a new rising edge at gearInAbsolute input
   END_STRUCT;
END_TYPE

TYPE "LAxisCtrl_typeGearInRelative"
TITLE = LAxisCtrl_typeGearInRelative
// Support: tech.team.motioncontrol@siemens.com 
// Fax: +49 (0) 9131/98-1297
   STRUCT
      ratioNumerator : DInt := 1;   // Gear ratio numerator
      ratioDenominator : DInt := 1;   // Gear ratio denominator
      acceleration : LReal := -1.0;   // Acceleration for synchronization (when "SyncProfileReference" = 0; Value > 0.0: The specified value is used; Value = 0.0: Not permitted; Value < 0.0: Use of the default value configured in the technology object)
      deceleration : LReal := -1.0;   // Deceleration for synchronization (when "SyncProfileReference" = 0; Value > 0.0: The specified value is used; Value = 0.0: Not permitted; Value < 0.0: Use of the default value configured in the technology object)
      jerk : LReal := -1.0;   // Jerk for synchronization (when "SyncProfileReference" = 0; Value > 0.0: Smooth velocity profile, the specified value is used; Value = 0.0: Trapezoid velocity profile; Value < 0.0: Use of the default value configured in the technology object)
      ratioChangeOnTheFly : Bool := FALSE;   // TRUE: Changing gear ratio on-the-fly; FALSE: Ratio change requires a new rising edge at gearInRelative input
   END_STRUCT;
END_TYPE

TYPE "LAxisCtrl_typeGeneralSettings"
TITLE = LAxisCtrl_typeGeneralSettings
// Support: tech.team.motioncontrol@siemens.com 
// Fax: +49 (0) 9131/98-1297
   STRUCT
      stopOnError : Bool := TRUE;   // TRUE: In case of error the axis will be stopped automatically with fastStop dynamics
      resetWithRestart : Bool := FALSE;   // TRUE: Reinitialization of the technology object and acknowledgment of pending technology alarms. The technology object is reinitialized with the configured start values; FALSE: Acknowledgment of queued technology alarms
      abortWaitingSyncCmd : Bool := TRUE;   // TRUE: Abort waiting synchronous command in case of new basic motion command automatically
   END_STRUCT;
END_TYPE

TYPE "LAxisCtrl_typeHoming"
TITLE = LAxisCtrl_typeHoming
// Support: tech.team.motioncontrol@siemens.com 
// Fax: +49 (0) 9131/98-1297
   STRUCT
      position : LReal := 0.0;   // The specified value is used according to the selected "Mode"
      mode : Int := 0;   // Operation mode; 0: Direct homing (absolute); 1:Direct homing (relative); 2:Passive homing (without reset); 3:Active homing; 5:Active homing (Position parameter has no effect); 6:Absolute encoder adjustment (relative); 7:Absolute encoder adjustment (absolute); 8:Passive homing ; 9:Abort passive homing; 10: Passive homing (Position parameter has no effect)
      extendedMode : DInt := -1;   // -1: No extended homing mode (parameter "mode" is effective); 0: Homing on fixed stop;
      extendedModeTorqueLimit : LReal := 0.0;   // Value of the torque/force for extended homing mode
   END_STRUCT;
END_TYPE

TYPE "LAxisCtrl_typeJog"
TITLE = LAxisCtrl_typeJog
// Support: tech.team.motioncontrol@siemens.com 
// Fax: +49 (0) 9131/98-1297
   STRUCT
      velocity : LReal := 0.0;   // Velocity for jogging (Value > 0.0: The specified value is used; Value = 0.0: Permitted; Value < 0.0: The absolute value of the specified value is used)
      acceleration : LReal := -1.0;   // Acceleration for jogging (Value > 0.0: The specified value is used; Value = 0.0: Not permitted; Value < 0.0: Use of the default value configured in the technology object)
      deceleration : LReal := -1.0;   // Deceleration for jogging (Value > 0.0: The specified value is used; Value = 0.0: Not permitted; Value < 0.0: Use of the default value configured in the technology object)
      jerk : LReal := -1.0;   // Jerk for jogging (Value > 0.0: Smooth velocity profile, the specified value is used; Value = 0.0: Trapezoid velocity profile; Value < 0.0: Use of the default value configured in the technology object)
      positionControlled : Bool := TRUE;   // TRUE: Position-controlled mode; FALSE: Non position-controlled operation
      increment : LReal := 0.0;   // Increment/distance for incremental jogging
      mode : DInt := 0;   // 0: Continuous jogging; 1: Incremental jogging new increment (starts with new increment); 2: Incremental jogging continue increment (continue the last increment if not completed)
   END_STRUCT;
END_TYPE

TYPE "LAxisCtrl_typeMoveVelocity"
TITLE = LAxisCtrl_typeMoveVelocity
// Support: tech.team.motioncontrol@siemens.com 
// Fax: +49 (0) 9131/98-1297
   STRUCT
      velocity : LReal := 0.0;   // Velocity/Speed for motion process (Value = 0.0: Permitted)
      acceleration : LReal := -1.0;   // Acceleration setpoint for motion process (Value > 0.0: The specified value is used; Value = 0.0: Not permitted; Value < 0.0: Use of the default value configured in the technology object)
      deceleration : LReal := -1.0;   // Deceleration setpoint for motion process (Value > 0.0: The specified value is used; Value = 0.0: Not permitted; Value < 0.0: Use of the default value configured in the technology object)
      jerk : LReal := -1.0;   // Jerk for velocity specification (Value > 0.0: Smooth velocity profile, the specified value is used; (Value = 0.0: Trapezoid velocity profile; (Value < 0.0: Use of the default value configured in the technology object)
      direction : Int := 0;   // Motion direction of the axis (0: The sign of the velocity parameter defines the direction; 1: Positive direction; 2: Negative direction)
      positionControlled : Bool := TRUE;   // TRUE: Position-controlled operation; FALSE: Non position-controlled operation
      velocityChangeOnTheFly : Bool := FALSE;   // TRUE: Changing velocity on-the-fly; FALSE: Velocity change requires a new rising edge on moveVelocity input
   END_STRUCT;
END_TYPE

TYPE "LAxisCtrl_typePhasing"
TITLE = LAxisCtrl_typePhasing
// Support: tech.team.motioncontrol@siemens.com 
// Fax: +49 (0) 9131/98-1297
   STRUCT
      phaseShift : LReal := 0.0;   // Absolute or relative leading value shift
      velocity : LReal := -1.0;   // Velocity for leading value shift, added to synchronous operation motion (Value > 0.0: The specified value is used; Value = 0.0: Not permitted; Value < 0.0: Use of the default value configured in the technology object)
      acceleration : LReal := -1.0;   // Acceleration for leading value shift, added to synchronous operation motion (Value > 0.0: The specified value is used; Value = 0.0: Not permitted; Value < 0.0: Use of the default value configured in the technology object)
      deceleration : LReal := -1.0;   // Deceleration for leading value shift, added to synchronous operation motion (Value > 0.0: The specified value is used; Value = 0.0: Not permitted; Value < 0.0: Use of the default value configured in the technology object)
      jerk : LReal := -1.0;   // Jerk for leading value shift, added to synchronous operation motion (Value > 0.0: Smooth velocity profile, the specified value is used; Value = 0.0: Trapezoid velocity profile; Value < 0.0: Use of the default value configured in the technology object)
      phaseAbsolute : Bool := TRUE;   // Indicates the type of phase shift. TRUE: Shift the leading value as an absolute shift; FALSE: Shift the leading value relative to the existing leading value shift
      phaseShiftChangeOnTheFly : Bool := FALSE;   // TRUE: Changing phase shift on-the-fly at absolute phasing; FALSE: Phase shift change requires a new rising edge at phasing input
   END_STRUCT;
END_TYPE

TYPE "LAxisCtrl_typePosAbsolute"
TITLE = LAxisCtrl_typePosAbsolute
// Support: tech.team.motioncontrol@siemens.com 
// Fax: +49 (0) 9131/98-1297
   STRUCT
      position : LReal := 0.0;   // Absolute target position
      velocity : LReal := -1.0;   // Velocity setpoint for absolute positioning (Value > 0.0: The specified value is used; Value = 0.0: Not permitted; Value < 0.0: Use of the default value configured in the technology object)
      acceleration : LReal := -1.0;   // Acceleration setpoint for absolute positioning (Value > 0.0: The specified value is used; Value = 0.0: Not permitted; Value < 0.0: Use of the default value configured in the technology object)
      deceleration : LReal := -1.0;   // Deceleration setpoint for absolute positioning (Value > 0.0: The specified value is used; Value = 0.0: Not permitted; Value < 0.0: Use of the default value configured in the technology object)
      jerk : LReal := -1.0;   // Jerk for absolute positioning (Value > 0.0: Smooth velocity profile, the specified value is used; (Value = 0.0: Trapezoid velocity profile; (Value < 0.0: Use of the default value configured in the technology object)
      direction : Int := 1;   // Motion direction of the axis (1: Positive direction; 2: Negative direction; 3: Shortest way)
      positionChangeOnTheFly : Bool := FALSE;   // TRUE: Changing position on-the-fly; FALSE: Position change requires a new rising edge at posAbsolute input
      velocityChangeOnTheFly : Bool := FALSE;   // TRUE: Changing velocity on-the-fly; FALSE: Velocity change requires a new rising edge at posAbsolute input
   END_STRUCT;
END_TYPE

TYPE "LAxisCtrl_typePosRelative"
TITLE = LAxisCtrl_typePosRelative
// Support: tech.team.motioncontrol@siemens.com 
// Fax: +49 (0) 9131/98-1297
   STRUCT
      distance : LReal := 0.0;   // Distance for positioning process
      velocity : LReal := -1.0;   // Velocity setpoint for relative positioning (Value > 0.0: The specified value is used; Value = 0.0: Not permitted; Value < 0.0: Use of the default value configured in the technology object)
      acceleration : LReal := -1.0;   // Acceleration setpoint for relative positioning (Value > 0.0: The specified value is used; Value = 0.0: Not permitted; Value < 0.0: Use of the default value configured in the technology object)
      deceleration : LReal := -1.0;   // Deceleration setpoint for relative positioning (Value > 0.0: The specified value is used; Value = 0.0: Not permitted; Value < 0.0: Use of the default value configured in the technology object)
      jerk : LReal := -1.0;   // Jerk for relative positioning (Value > 0.0: Smooth velocity profile, the specified value is used; Value = 0.0: Trapezoid velocity profile; Value < 0.0: Use of the default value configured in the technology object)
      direction : DInt := 0;   // Motion direction of the axis (0: The sign of the distance parameter defines the direction; 1: Positive direction; 2: Negative direction)
   END_STRUCT;
END_TYPE

TYPE "LAxisCtrl_typePosSuperimposed"
TITLE = LAxisCtrl_typePosSuperimposed
// Support: tech.team.motioncontrol@siemens.com 
// Fax: +49 (0) 9131/98-1297
   STRUCT
      distance : LReal := 0.0;   // Distance for superimposed positioning
      velocityDiff : LReal := -1.0;   // Maximum velocity deviation compared to the active motion (Value > 0.0: The specified value is used; Value = 0.0: Not permitted; Value < 0.0: Use of the default value configured in the technology object)
      acceleration : LReal := -1.0;   // Acceleration for positioning (Value > 0.0: The specified value is used; Value = 0.0: Not permitted; Value < 0.0: Use of the default value configured in the technology object)
      deceleration : LReal := -1.0;   // Deceleration for positioning (Value > 0.0: The specified value is used; Value = 0.0: Not permitted; Value < 0.0: Use of the default value configured in the technology object)
      jerk : LReal := -1.0;   // Jerk for positioning (Value > 0.0: Smooth velocity profile, the specified value is used; Value = 0.0: Trapezoid velocity profile; Value < 0.0: Use of the default value configured in the technology object)
      direction : DInt := 0;   // Motion direction of the axis (0: The sign of the distance parameter defines the direction; 1: Positive negative; 2: Negative direction)
   END_STRUCT;
END_TYPE

TYPE "LAxisCtrl_typePower"
TITLE = LAxisCtrl_typePower
// Support: tech.team.motioncontrol@siemens.com 
// Fax: +49 (0) 9131/98-1297
   STRUCT
      startMode : DInt := 1;   // 0: Enable axis not position-controlled; 1: Enable axis position-controlled (This parameter is ignored when a speed axis or external encoder is used)
      stopMode : Int := 0;   // 0: Emergency stop; 1: Immediate stop; 2: Stop with maximum dynamic values
      syncMotionSimulation : Bool := FALSE;   // TRUE: Start the simulation of synchronous operation automatically with falling edge at enableAxis; FALSE: No simulation of synchronous operation
   END_STRUCT;
END_TYPE

TYPE "LAxisCtrl_typeStop"
TITLE = LAxisCtrl_typeStop
// Support: tech.team.motioncontrol@siemens.com 
// Fax: +49 (0) 9131/98-1297
   STRUCT
      deceleration : LReal := -1.0;   // Deceleration setpoint for stop (Value > 0.0: The specified value is used; Value = 0.0: Not permitted; Value < 0.0: Use of the default value configured in the technology object)
      jerk : LReal := -1.0;   // Jerk for stop (Value > 0.0: Smooth velocity profile, the specified value is used; Value = 0.0: Trapezoid velocity profile; Value < 0.0: Use of the default value configured in the technology object)
      abortAcceleration : Bool := FALSE;   // TRUE: The acceleration is set to 0.0 at the start of the job, and the deceleration immediately builds up; FALSE: The current acceleration at the start of the job is reduced using the configured jerk. Afterwards, the deceleration builds up
   END_STRUCT;
END_TYPE

TYPE "LAxisCtrl_typeTorqueLimiting"
TITLE = LAxisCtrl_typeTorqueLimiting
// Support: tech.team.motioncontrol@siemens.com 
// Fax: +49 (0) 9131/98-1297
   STRUCT
      limit : LReal := -1.0;   // Value of force/torque limiting (in the configured unit of measurement)
      mode : DInt := 0;   // 0: Force/Torque limiting; 1: Fixed stop detection
   END_STRUCT;
END_TYPE

DATA_BLOCK "HMI变量汇总"   // DB10
{ S7_Optimized_Access := 'TRUE' }
// stored: MemoryReserve 100
   VAR
      Vis_Button_wideX1 : Bool;
      Vis_Button_wideX2 : Bool;
      Vis_Button_wideX3 : Bool;
      Vis_Button_wideX4 : Bool;
      Vis_Button_wideX5 : Bool;
      Vis_Button_wideX6 : Bool;
      Vis_Button_wideX7 : Bool;
      Vis_Button_wideX8 : Bool;
      Vis_Button_wideX9 : Bool;
      Vis_Button_wideX10 : Bool;
      Vis_Button_wideX11 : Bool;
      Vis_Button_wideX12 : Bool;
      Vis_Button_small1 : Bool;
      Vis_Button_small2 : Bool;
      Vis_Button_small3 : Bool;
      Vis_Button_small4 : Bool;
      Vis_Button_small5 : Bool;
      Vis_Button_small6 : Bool;
      Vis_Button_small7 : Bool;
      Vis_Button_small8 : Bool;
      Vis_Button_small9 : Bool;
      Vis_Button_small10 : Bool;
      Vis_Button_small11 : Bool;
      Vis_Button_small12 : Bool;
   END_VAR
BEGIN
END_DATA_BLOCK

DATA_BLOCK "气缸面板多路复用变量"   // DB11
{ S7_Optimized_Access := 'TRUE' }
// stored: MemoryReserve 100
   VAR
      Valve_index : "VALVE_HMI_UDT";
      HMI_Positon_X24 { S7_SetPoint := 'True'} : Bool;
   END_VAR
BEGIN
END_DATA_BLOCK

DATA_BLOCK "PN_DEV_DIAG_PD_DB"   // DB100
{ S7_Optimized_Access := 'TRUE' }
// stored: AutoNumber false, MemoryReserve 100
   VAR
      DEVICE_DATA : "PN_DEV_DIAG_STRUCT_UDT";
   END_VAR
BEGIN
END_DATA_BLOCK

DATA_BLOCK "EQUIPMENT_DATA_GLOBAL_DB"   // DB200
{ S7_Optimized_Access := 'TRUE' }
// stored: AutoNumber false, MemoryReserve 100
   VAR RETAIN
      EmptyStepHistory { S7_SetPoint := 'True'} : Array[0.."EQUIPMENTDATA_STEPHISTORYLENGTH"] of "GRAPH_STEP_HISTORY_UDT";
   END_VAR
   VAR
      Dummy_IF_COND { ExternalAccessible := 'False'; ExternalVisible := 'False'; ExternalWritable := 'False'; S7_SetPoint := 'True'} : "COND_PD_UDT";
   END_VAR
BEGIN
END_DATA_BLOCK

DATA_BLOCK "EQUIPMENT_DATA_SCADA_DB"   // DB201
{ S7_Optimized_Access := 'TRUE' }
// stored: AutoNumber false, MemoryReserve 100
   VAR
      PLC1_OPMODE01 { ExternalWritable := 'False'} : "EQUIPMENT_DATA_OUT_UDT";
      PLC1_OPMODE02 { ExternalWritable := 'False'} : "EQUIPMENT_DATA_OUT_UDT";
      PLC1_OPMODE03 { ExternalWritable := 'False'} : "EQUIPMENT_DATA_OUT_UDT";
      PLC1_OPMODE04 { ExternalWritable := 'False'} : "EQUIPMENT_DATA_OUT_UDT";
      PLC1_OPMODE05 { ExternalWritable := 'False'} : "EQUIPMENT_DATA_OUT_UDT";
      PLC1_OPMODE06 { ExternalWritable := 'False'} : "EQUIPMENT_DATA_OUT_UDT";
      PLC1_OPMODE01_ST010 { ExternalWritable := 'False'} : "EQUIPMENT_DATA_OUT_UDT";
      PLC1_OPMODE02_Buffer { ExternalWritable := 'False'} : "EQUIPMENT_DATA_OUT_UDT";
      PLC1_OPMODE03_Buffer { ExternalWritable := 'False'} : "EQUIPMENT_DATA_OUT_UDT";
      PLC1_OPMODE04_Buffer { ExternalWritable := 'False'} : "EQUIPMENT_DATA_OUT_UDT";
      PLC1_OPMODE05_ST020 { ExternalWritable := 'False'} : "EQUIPMENT_DATA_OUT_UDT";
      PLC1_OPMODE06_ST025 { ExternalWritable := 'False'} : "EQUIPMENT_DATA_OUT_UDT";
      PLC1_OPMODE06_ST030 { ExternalWritable := 'False'} : "EQUIPMENT_DATA_OUT_UDT";
      PLC1_OPMODE06_ST035 { ExternalWritable := 'False'} : "EQUIPMENT_DATA_OUT_UDT";
      TEST_EqtData { ExternalWritable := 'False'} : "EQUIPMENT_DATA_OUT_UDT";
   END_VAR
BEGIN
END_DATA_BLOCK

DATA_BLOCK "GLOBAL_Axis_HMI_IF_DB"   // DB202
{ S7_Optimized_Access := 'TRUE' }
// stored: AutoNumber false, MemoryReserve 100
   VAR RETAIN
      Axis { S7_SetPoint := 'True'} : Array[0..20] of "Axis_IF_HMI";
   END_VAR
BEGIN
END_DATA_BLOCK

DATA_BLOCK "GLOBAL_DRIVE_HMI_IF_DB"   // DB203
{ S7_Optimized_Access := 'TRUE' }
AUTHOR : Tesla
FAMILY : Drive
VERSION : 1.0
// stored: AutoNumber false, MemoryReserve 100
   VAR RETAIN
      Drive : Array[0.."No_Drives"] of "DRIVE_HMI_UDT";
   END_VAR
BEGIN
END_DATA_BLOCK

DATA_BLOCK "GLOBAL_G120D_RBD_HMI_IF_DB"   // DB204
{ S7_Optimized_Access := 'TRUE' }
// stored: AutoNumber false, MemoryReserve 100
   VAR RETAIN
      RBD { S7_SetPoint := 'True'} : Array[0..10] of "H_HMI";
   END_VAR
   VAR
      RBD_G120D { S7_SetPoint := 'True'} : Array[0..6] of "H_Roller2W2S-G120PN";
   END_VAR
BEGIN
   // RBD[1] : ST010RBD01
   // RBD[2] : ST020RBD01
   // RBD[5] : ST030RBD01
   // RBD[6] : ST035RBD01
   // RBD_G120D[1] : ST010RBD01
   // RBD_G120D[2] : ST020RBD01
   // RBD_G120D[5] : ST030RBD01
   // RBD_G120D[6] : ST035RBD01
END_DATA_BLOCK

DATA_BLOCK "GLOBAL_GRAPH_HMI_IF_DB"   // DB205
{ S7_Optimized_Access := 'TRUE' }
// stored: AutoNumber false, MemoryReserve 100
   VAR
      GRAPH : Array[0..20] of "GRAPH_CONTROL_UDT";
   END_VAR
BEGIN
   // GRAPH[1] : ST010_MAIN_GRAPH_FB
   // GRAPH[2] : ST020_CNV06_GRAPH_FB
   // GRAPH[3] : ST020_CNV04_GRAPH_FB
   // GRAPH[4] : ST020_CNV05_GRAPH_FB
   // GRAPH[5] : ST020_MAIN_GRAPH_FB
   // GRAPH[6] : ST020_ROBOT_GRAPH_FB
   // GRAPH[7] : ST020_RB01_GRAPH_FB
   // GRAPH[8] : ST020_RB02_GRAPH_FB
   // GRAPH[9] : ST020_RB06_GRAPH_FB
   // GRAPH[10] : ST025_RB01_GRAPH_FB
   // GRAPH[11] : ST025_RB02_GRAPH_FB
   // GRAPH[12] : ST025_TL01_GRAPH_FB
   // GRAPH[13] : ST025_TL02_GRAPH_FB
   // GRAPH[14] : ST030_MAIN_GRAPH_FB
   // GRAPH[15] : ST030_ROBOT_GRAPH_FB
   // GRAPH[16] : ST030_SLIDE_GRAPH_FB
   // GRAPH[17] : ST035_MAIN_GRAPH_FB
END_DATA_BLOCK

DATA_BLOCK "GLOBAL_HMI_SCREEN_NO_IF_DB"   // DB206
{ S7_Optimized_Access := 'TRUE' }
// stored: AutoNumber false, MemoryReserve 100
   VAR
      HMI : Array[0..1] of "HMI_SCREEN_NO_AREA_POINTER_UDT";
   END_VAR
BEGIN
END_DATA_BLOCK

DATA_BLOCK "GLOBAL_IDENT_DATA_DB"   // DB207
{ S7_Optimized_Access := 'TRUE' }
AUTHOR : Tesla
FAMILY : Ident
VERSION : 1.0
// stored: AutoNumber false, MemoryReserve 100
   VAR
      Reader { ExternalAccessible := 'False'; ExternalVisible := 'False'; ExternalWritable := 'False'; S7_SetPoint := 'True'} : Array[0.."No_Reader"] of "IDENT_RW_BYTE_DAT_UDT";
   END_VAR
BEGIN
END_DATA_BLOCK

DATA_BLOCK "GLOBAL_IDENT_HMI_IF_DB"   // DB208
{ S7_Optimized_Access := 'TRUE' }
AUTHOR : Tesla
FAMILY : Ident
VERSION : 1.0
// stored: AutoNumber false, MemoryReserve 100
   VAR
      Reader { S7_SetPoint := 'True'} : Array[0.."No_Reader"] of "IDENT_RW_HMI_DAT_UDT";   // Data Erased On Tag Not Present / 数据 Erased 打开 Tag 没有 在
   END_VAR
BEGIN
END_DATA_BLOCK

DATA_BLOCK "GLOBAL_PP_HMI_IF_DB"   // DB210
{ S7_Optimized_Access := 'TRUE' }
// stored: AutoNumber false, MemoryReserve 100
   VAR
      PP : Array[0..200] of "TEC_UNIT_HMI_UDT";
      Hide_PP_Check : Array[0..200] of Bool;
      Check_TON : Array[0..200] of TON_TIME;
   END_VAR
BEGIN
   // PP[0] : 放卷上位
   // PP[1] : +ST020-CNV06-VM01-PX01 / 放卷下位
   // PP[2] : +ST020-CNV06-VM01-PX02 / +ST010-TL02- PP01
   // PP[3] : +ST020-CNV06-VM01-PX03 / +ST010-TL02- PP02
   // PP[4] : +ST020-TL01- PP01
   // PP[5] : +ST020-CNV06-VM01-PX05 / +ST020-TL01- PP02
   // PP[6] : +ST020-CNV06-VM01-PX06 / +ST020-TL02- PP01
   // PP[7] : +ST020-CNV06-VM01-PX07 / +ST020-TL02- PP02
   // PP[8] : +ST020-CNV06-VM01-PX08
   // PP[9] : +ST020-CNV06-VM01-PX09
   // PP[10] : +ST020-CNV06-VM01-PX10
   // PP[11] : +ST020-CNV06-VM01-PX11
   // PP[12] : +ST020-CNV06-VM01-PX20
   // PP[13] : +ST020-CNV06-VM01-PEY01
   // PP[14] : +ST020-CNV06-VM01-PEY02
   // PP[15] : +ST020-CNV06-VM01-PEY03
   // PP[16] : +ST020-CNV06-VM01-PEY04
   // PP[17] : +ST020-CNV06-PX21
   // PP[18] : +ST020-CNV06-PX12
   // PP[20] : +ST020-CNV04-VM01-PX01 Unload Pos1
   // PP[21] : +ST020-CNV04-VM01-PX02 Unload Pos2
   // PP[22] : +ST020-CNV04-VM01-PX03 Unload Pos3
   // PP[23] : +ST020-CNV04-VM01-PX04 WaitPos1 Off
   // PP[24] : +ST020-CNV04-VM01-PX05 WaitPos1
   // PP[25] : +ST020-CNV04-VM01-PX06 WaitPos2 Off
   // PP[26] : +ST020-CNV04-VM01-PX07 WaitPos2
   // PP[27] : +ST020-CNV04-VM01-PX08 WaitPos2 Full
   // PP[28] : +ST020-CNV04-VM01-PX09 WaitPos3 Off
   // PP[29] : +ST020-CNV04-VM01-PX10 WaitPos3
   // PP[30] : +ST020-CNV04-VM01-PX11 WaitPos3 Full
   // PP[31] : +ST020-CNV04-VM01-PX12 WaitPos4 Off
   // PP[32] : +ST020-CNV04-VM01-PX13 WaitPos4
   // PP[33] : +ST020-CNV04-VM01-PX17 LoadPos Off
   // PP[34] : +ST020-CNV04-VM01-PX14 LoadPos1
   // PP[35] : +ST020-CNV04-VM01-PX15 LoadPos2
   // PP[36] : +ST020-CNV04-VM01-PX16 LoadPos3
   // PP[37] : +ST020-CNV04-VM01-PX19 LoadPos4
   // PP[38] : +ST020-CNV04-VM01-PX18 LoadposBypass
   // PP[39] : +ST020-CNV04-VM01-PX20 LoadPos Ready
   // PP[40] : +ST020-CNV04-VM01-PX21 Unload Pos
   // PP[41] : +ST020-CNV04-VM01-PX36 Chain Check
   // PP[42] : +ST020-CNV04-VM01-PX37 Load Slide Table Check
   // PP[43] : +ST020-CNV04-VM01-PX38 Unload Slide Table Check
   // PP[44] : +ST020-CNV04-VM01-PEY01 Unload Part Check
   // PP[45] : +ST020-CNV04-VM01-PEY02 Unload Part Check
   // PP[46] : +ST020-CNV04-VM01-PEY03 Load Part Check
   // PP[47] : +ST020-CNV04-VM01-PEY04 Load Part Check
   // PP[48] : +ST020-CNV04-VM01-PX22 Unload Pos Full
   // PP[50] : +ST020-TL12-SX02
   // PP[51] : +ST020-CNV05-VM01-PX01
   // PP[52] : +ST020-CNV05-VM01-PX02
   // PP[53] : +ST020-CNV05-VM01-PX03
   // PP[54] : +ST020-CNV05-VM01-PX04
   // PP[55] : +ST020-CNV05-VM01-PX05
   // PP[56] : +ST020-CNV05-VM01-PX06
   // PP[57] : +ST020-CNV05-VM01-PX07
   // PP[58] : +ST020-CNV05-VM01-PX08
   // PP[59] : +ST020-CNV05-VM01-PX09
   // PP[60] : +ST020-CNV05-VM01-PX11
   // PP[61] : +ST020-CNV05-VM01-PX10
   // PP[62] : +ST020-CNV05-VM01-PX12
   // PP[63] : +ST020-CNV05-VM01-PX13
   // PP[64] : +ST020-CNV05-VM01-PX14
   // PP[65] : +ST020-CNV05-VM01-PX15
   // PP[66] : +ST020-CNV05-VM01-PX16
   // PP[67] : +ST020-CNV05-VM01-PX17
   // PP[68] : +ST020-CNV05-VM01-PX19
   // PP[69] : +ST020-CNV05-VM01-PX20
   // PP[70] : +ST020-CNV05-VM01-PX25
   // PP[71] : +ST020-CNV05-VM01-PX21
   // PP[72] : +ST020-CNV05-VM01-PX22
   // PP[73] : +ST020-CNV05-VM01-PX23
   // PP[74] : +ST020-CNV05-PX40
   // PP[75] : +ST020-CNV05-PX41
   // PP[76] : +ST020-CNV05-PX42
   // PP[77] : +ST020-CNV05-PEY01
   // PP[78] : +ST020-CNV05-PEY02
   // PP[79] : +ST020-CNV05-PEY03
   // PP[80] : +ST020-CNV05-PEY04
   // PP[81] : +ST020-TL01-PX01
   // PP[82] : +ST020-TL01-PX02
   // PP[83] : +ST020-TL01-PX03
   // PP[84] : +ST020-TL01-PX04
   // PP[85] : +ST020-TL01-PX05
   // PP[86] : +ST020-TL01-PX06
   // PP[87] : +ST020-TL01-PX07
   // PP[88] : +ST020-TL01-PX08
   // PP[89] : +ST020-TL01-PX09
   // PP[90] : +ST020-TL01-PX10
   // PP[91] : +ST020-TO01-PEY01
   // PP[92] : +ST020-TL09-SX01
   // PP[93] : +ST020-TL09-SX02
   // PP[94] : +ST020-TO02-PEY01
   // PP[95] : +ST020-TL10-SX01
   // PP[96] : +ST020-TL10-SX02
   // PP[97] : +ST020-TO04-PEY01
   // PP[98] : +ST020-TO04-PEY02
   // PP[99] : +ST020-TL12-SX01
   // PP[100] : +ST025-TL01- PX01
   // PP[101] : +ST025-TL01- PX02
   // PP[102] : +ST025-TL01- PX03
   // PP[103] : +ST025-TL01- PX04
   // PP[104] : +ST025-TL02- PX01
   // PP[105] : +ST025-TL02- PX02
   // PP[106] : +ST025-TL02- PX03
   // PP[107] : +ST025-TL02- PX04
   // PP[108] : +ST030-TL01- PX01
   // PP[109] : +ST030-TL01- PX02
   // PP[110] : +ST030-TL01- PX03
   // PP[111] : +ST030-TL01- PX04
   // PP[112] : +ST030-TL01- PX05
   // PP[113] : +ST030-TL01- PX06
   // PP[114] : +ST030-TL01- PX07
   // PP[115] : +ST030-TL01- PX08
   // PP[116] : +ST030-TL01- PX09
   // PP[117] : +ST030-TL01- PX10
   // PP[118] : +ST030-TL03- PX01
   // PP[119] : +ST030-TL03- PX02
   // PP[120] : +ST030-TL04- PX01
   // PP[121] : +ST030-TL04- PX02
   // PP[122] : +ST010-PX01
   // PP[123] : +ST010-PX02
   // PP[124] : +ST030-TL01- PX11
   // PP[125] : +ST010-OffLine_PX01
   // PP[126] : +ST010-OffLine_PX02
   // PP[127] : ST020_LFT01_Repair
   // PP[128] : ST030_LFT01_Repair
   // PP[129] : ST035_LFT01_Repair
   // PP[130] : +ST020-CNV0-PX39 TakeposBypass
   // PP[131] : +ST030-TL03- PX03
   // PP[132] : +ST030-TL03- PX04
   // PP[133] : +ST030-TL04- PX03
   // PP[134] : +ST030-TL04- PX04
   // PP[135] : +ST020-CNV05-PX26
   // PP[136] : +ST010RBD01--PX04(OverSensor)
   // PP[137] : +ST020RBD01--PX04(OverSensor)
   // PP[138] : +ST030RBD01--PX04(OverSensor)
   // PP[139] : +ST035RBD01--PX04(OverSensor)
   // PP[140] : ST010PSW01
   // PP[141] : "+ST020-TL01-VM01-PSW01"
   // PP[142] : "+ST020-TL09-VM01-PSW01"
   // PP[143] : "+ST020-TL10-VM01-PSW01"
   // PP[144] : "+ST025-TL01-VM01-PSW01"
   // PP[145] : "+ST025-TL02-VM01-PSW01"
   // PP[146] : "+ST030-TL01-VM01-PSW01"
   // Hide_PP_Check[1] : +ST020-CNV06-VM01-PX01
   // Hide_PP_Check[2] : +ST020-CNV06-VM01-PX02
   // Hide_PP_Check[3] : +ST020-CNV06-VM01-PX03
   // Hide_PP_Check[5] : +ST020-CNV06-VM01-PX05
   // Hide_PP_Check[6] : +ST020-CNV06-VM01-PX06
   // Hide_PP_Check[7] : +ST020-CNV06-VM01-PX07
   // Hide_PP_Check[8] : +ST020-CNV06-VM01-PX08
   // Hide_PP_Check[9] : +ST020-CNV06-VM01-PX09
   // Hide_PP_Check[10] : +ST020-CNV06-VM01-PX10
   // Hide_PP_Check[11] : +ST020-CNV06-VM01-PX11
   // Hide_PP_Check[12] : +ST020-CNV06-VM01-PX20
   // Hide_PP_Check[13] : +ST020-CNV06-VM01-PEY01
   // Hide_PP_Check[14] : +ST020-CNV06-VM01-PEY02
   // Hide_PP_Check[15] : +ST020-CNV06-VM01-PEY03
   // Hide_PP_Check[16] : +ST020-CNV06-VM01-PEY04
   // Hide_PP_Check[17] : +ST020-CNV06-PX21
   // Hide_PP_Check[20] : +ST020-CNV04-VM01-PX01 Unload Pos1
   // Hide_PP_Check[21] : +ST020-CNV04-VM01-PX02 Unload Pos2
   // Hide_PP_Check[22] : +ST020-CNV04-VM01-PX03 Unload Pos3
   // Hide_PP_Check[23] : +ST020-CNV04-VM01-PX04 WaitPos1 Off
   // Hide_PP_Check[24] : +ST020-CNV04-VM01-PX05 WaitPos1
   // Hide_PP_Check[25] : +ST020-CNV04-VM01-PX06 WaitPos2 Off
   // Hide_PP_Check[26] : +ST020-CNV04-VM01-PX07 WaitPos2
   // Hide_PP_Check[27] : +ST020-CNV04-VM01-PX08 WaitPos2 Full
   // Hide_PP_Check[28] : +ST020-CNV04-VM01-PX09 WaitPos3 Off
   // Hide_PP_Check[29] : +ST020-CNV04-VM01-PX10 WaitPos3
   // Hide_PP_Check[30] : +ST020-CNV04-VM01-PX11 WaitPos3 Full
   // Hide_PP_Check[31] : +ST020-CNV04-VM01-PX12 WaitPos4 Off
   // Hide_PP_Check[32] : +ST020-CNV04-VM01-PX13 WaitPos4
   // Hide_PP_Check[33] : +ST020-CNV04-VM01-PX17 LoadPos Off
   // Hide_PP_Check[34] : +ST020-CNV04-VM01-PX14 LoadPos1
   // Hide_PP_Check[35] : +ST020-CNV04-VM01-PX15 LoadPos2
   // Hide_PP_Check[36] : +ST020-CNV04-VM01-PX16 LoadPos3
   // Hide_PP_Check[37] : +ST020-CNV04-VM01-PX19 LoadPos4
   // Hide_PP_Check[38] : +ST020-CNV04-VM01-PX18 LoadposBypass
   // Hide_PP_Check[39] : +ST020-CNV04-VM01-PX20 LoadPos Ready
   // Hide_PP_Check[40] : +ST020-CNV04-VM01-PX21 Unload Pos
   // Hide_PP_Check[41] : +ST020-CNV04-VM01-PX36 Chain Check
   // Hide_PP_Check[42] : +ST020-CNV04-VM01-PX37 Load Slide Table Check
   // Hide_PP_Check[43] : +ST020-CNV04-VM01-PX38 Unload Slide Table Check
   // Hide_PP_Check[44] : +ST020-CNV04-VM01-PEY01 Unload Part Check
   // Hide_PP_Check[45] : +ST020-CNV04-VM01-PEY02 Unload Part Check
   // Hide_PP_Check[46] : +ST020-CNV04-VM01-PEY03 Load Part Check
   // Hide_PP_Check[47] : +ST020-CNV04-VM01-PEY04 Load Part Check
   // Hide_PP_Check[48] : +ST020-CNV04-VM01-PX22 Unload Pos Full
   // Hide_PP_Check[50] : +ST020-TL12-SX02
   // Hide_PP_Check[51] : +ST020-CNV05-VM01-PX01
   // Hide_PP_Check[52] : +ST020-CNV05-VM01-PX02
   // Hide_PP_Check[53] : +ST020-CNV05-VM01-PX03
   // Hide_PP_Check[54] : +ST020-CNV05-VM01-PX04
   // Hide_PP_Check[55] : +ST020-CNV05-VM01-PX05
   // Hide_PP_Check[56] : +ST020-CNV05-VM01-PX06
   // Hide_PP_Check[57] : +ST020-CNV05-VM01-PX07
   // Hide_PP_Check[58] : +ST020-CNV05-VM01-PX08
   // Hide_PP_Check[59] : +ST020-CNV05-VM01-PX09
   // Hide_PP_Check[60] : +ST020-CNV05-VM01-PX11
   // Hide_PP_Check[61] : +ST020-CNV05-VM01-PX10
   // Hide_PP_Check[62] : +ST020-CNV05-VM01-PX12
   // Hide_PP_Check[63] : +ST020-CNV05-VM01-PX13
   // Hide_PP_Check[64] : +ST020-CNV05-VM01-PX14
   // Hide_PP_Check[65] : +ST020-CNV05-VM01-PX15
   // Hide_PP_Check[66] : +ST020-CNV05-VM01-PX16
   // Hide_PP_Check[67] : +ST020-CNV05-VM01-PX17
   // Hide_PP_Check[68] : +ST020-CNV05-VM01-PX19
   // Hide_PP_Check[69] : +ST020-CNV05-VM01-PX20
   // Hide_PP_Check[70] : +ST020-CNV05-VM01-PX25
   // Hide_PP_Check[71] : +ST020-CNV05-VM01-PX21
   // Hide_PP_Check[72] : +ST020-CNV05-VM01-PX22
   // Hide_PP_Check[73] : +ST020-CNV05-VM01-PX23
   // Hide_PP_Check[74] : +ST020-CNV05-PX40
   // Hide_PP_Check[75] : +ST020-CNV05-PX41
   // Hide_PP_Check[76] : +ST020-CNV05-PX42
   // Hide_PP_Check[77] : +ST020-CNV05-PEY01
   // Hide_PP_Check[78] : +ST020-CNV05-PEY02
   // Hide_PP_Check[79] : +ST020-CNV05-PEY03
   // Hide_PP_Check[80] : +ST020-CNV05-PEY04
   // Hide_PP_Check[81] : +ST020-TL01-PX01
   // Hide_PP_Check[82] : +ST020-TL01-PX02
   // Hide_PP_Check[83] : +ST020-TL01-PX03
   // Hide_PP_Check[84] : +ST020-TL01-PX04
   // Hide_PP_Check[85] : +ST020-TL01-PX05
   // Hide_PP_Check[86] : +ST020-TL01-PX06
   // Hide_PP_Check[87] : +ST020-TL01-PX07
   // Hide_PP_Check[88] : +ST020-TL01-PX08
   // Hide_PP_Check[89] : +ST020-TL01-PX09
   // Hide_PP_Check[90] : +ST020-TL01-PX10
   // Hide_PP_Check[91] : +ST020-TO01-PEY01
   // Hide_PP_Check[92] : +ST020-TL09-SX01
   // Hide_PP_Check[93] : +ST020-TL09-SX02
   // Hide_PP_Check[94] : +ST020-TO02-PEY01
   // Hide_PP_Check[95] : +ST020-TL10-SX01
   // Hide_PP_Check[96] : +ST020-TL10-SX02
   // Hide_PP_Check[97] : +ST020-TO04-PEY01
   // Hide_PP_Check[98] : +ST020-TO04-PEY02
   // Hide_PP_Check[99] : +ST020-TL12-SX01
   // Hide_PP_Check[100] : +ST025-TL01- PX01
   // Hide_PP_Check[101] : +ST025-TL01- PX02
   // Hide_PP_Check[102] : +ST025-TL01- PX03
   // Hide_PP_Check[103] : +ST025-TL01- PX04
   // Hide_PP_Check[104] : +ST025-TL02- PX01
   // Hide_PP_Check[105] : +ST025-TL02- PX02
   // Hide_PP_Check[106] : +ST025-TL02- PX03
   // Hide_PP_Check[107] : +ST025-TL02- PX04
   // Hide_PP_Check[108] : +ST030-TL01- PX01
   // Hide_PP_Check[109] : +ST030-TL01- PX02
   // Hide_PP_Check[110] : +ST030-TL01- PX03
   // Hide_PP_Check[111] : +ST030-TL01- PX04
   // Hide_PP_Check[112] : +ST030-TL01- PX05
   // Hide_PP_Check[113] : +ST030-TL01- PX06
   // Hide_PP_Check[114] : +ST030-TL01- PX07
   // Hide_PP_Check[115] : +ST030-TL01- PX08
   // Hide_PP_Check[116] : +ST030-TL01- PX09
   // Hide_PP_Check[117] : +ST030-TL01- PX10
   // Hide_PP_Check[118] : +ST030-TL03- PX01
   // Hide_PP_Check[119] : +ST030-TL03- PX02
   // Hide_PP_Check[120] : +ST030-TL04- PX01
   // Hide_PP_Check[121] : +ST030-TL04- PX02
   // Hide_PP_Check[122] : +ST010-PX01
   // Hide_PP_Check[123] : +ST010-PX02
   // Hide_PP_Check[124] : +ST030-TL01- PX11
   // Hide_PP_Check[125] : +ST010-OffLine_PX01
   // Hide_PP_Check[126] : +ST010-OffLine_PX02
   // Hide_PP_Check[127] : ST020_LFT01_Repair
   // Hide_PP_Check[128] : ST030_LFT01_Repair
   // Hide_PP_Check[129] : ST035_LFT01_Repair
   // Hide_PP_Check[130] : +ST020-CNV0-PX39 TakeposBypass
   // Hide_PP_Check[131] : +ST030-TL03- PX03
   // Hide_PP_Check[132] : +ST030-TL03- PX04
   // Hide_PP_Check[133] : +ST030-TL04- PX03
   // Hide_PP_Check[134] : +ST030-TL04- PX04
   // Check_TON[1] : +ST020-CNV06-VM01-PX01
   // Check_TON[2] : +ST020-CNV06-VM01-PX02
   // Check_TON[3] : +ST020-CNV06-VM01-PX03
   // Check_TON[5] : +ST020-CNV06-VM01-PX05
   // Check_TON[6] : +ST020-CNV06-VM01-PX06
   // Check_TON[7] : +ST020-CNV06-VM01-PX07
   // Check_TON[8] : +ST020-CNV06-VM01-PX08
   // Check_TON[9] : +ST020-CNV06-VM01-PX09
   // Check_TON[10] : +ST020-CNV06-VM01-PX10
   // Check_TON[11] : +ST020-CNV06-VM01-PX11
   // Check_TON[12] : +ST020-CNV06-VM01-PX20
   // Check_TON[13] : +ST020-CNV06-VM01-PEY01
   // Check_TON[14] : +ST020-CNV06-VM01-PEY02
   // Check_TON[15] : +ST020-CNV06-VM01-PEY03
   // Check_TON[16] : +ST020-CNV06-VM01-PEY04
   // Check_TON[17] : +ST020-CNV06-PX21
   // Check_TON[20] : +ST020-CNV04-VM01-PX01 Unload Pos1
   // Check_TON[21] : +ST020-CNV04-VM01-PX02 Unload Pos2
   // Check_TON[22] : +ST020-CNV04-VM01-PX03 Unload Pos3
   // Check_TON[23] : +ST020-CNV04-VM01-PX04 WaitPos1 Off
   // Check_TON[24] : +ST020-CNV04-VM01-PX05 WaitPos1
   // Check_TON[25] : +ST020-CNV04-VM01-PX06 WaitPos2 Off
   // Check_TON[26] : +ST020-CNV04-VM01-PX07 WaitPos2
   // Check_TON[27] : +ST020-CNV04-VM01-PX08 WaitPos2 Full
   // Check_TON[28] : +ST020-CNV04-VM01-PX09 WaitPos3 Off
   // Check_TON[29] : +ST020-CNV04-VM01-PX10 WaitPos3
   // Check_TON[30] : +ST020-CNV04-VM01-PX11 WaitPos3 Full
   // Check_TON[31] : +ST020-CNV04-VM01-PX12 WaitPos4 Off
   // Check_TON[32] : +ST020-CNV04-VM01-PX13 WaitPos4
   // Check_TON[33] : +ST020-CNV04-VM01-PX17 LoadPos Off
   // Check_TON[34] : +ST020-CNV04-VM01-PX14 LoadPos1
   // Check_TON[35] : +ST020-CNV04-VM01-PX15 LoadPos2
   // Check_TON[36] : +ST020-CNV04-VM01-PX16 LoadPos3
   // Check_TON[37] : +ST020-CNV04-VM01-PX19 LoadPos4
   // Check_TON[38] : +ST020-CNV04-VM01-PX18 LoadposBypass
   // Check_TON[39] : +ST020-CNV04-VM01-PX20 LoadPos Ready
   // Check_TON[40] : +ST020-CNV04-VM01-PX21 Unload Pos
   // Check_TON[41] : +ST020-CNV04-VM01-PX36 Chain Check
   // Check_TON[42] : +ST020-CNV04-VM01-PX37 Load Slide Table Check
   // Check_TON[43] : +ST020-CNV04-VM01-PX38 Unload Slide Table Check
   // Check_TON[44] : +ST020-CNV04-VM01-PEY01 Unload Part Check
   // Check_TON[45] : +ST020-CNV04-VM01-PEY02 Unload Part Check
   // Check_TON[46] : +ST020-CNV04-VM01-PEY03 Load Part Check
   // Check_TON[47] : +ST020-CNV04-VM01-PEY04 Load Part Check
   // Check_TON[48] : +ST020-CNV04-VM01-PX22 Unload Pos Full
   // Check_TON[50] : +ST020-TL12-SX02
   // Check_TON[51] : +ST020-CNV05-VM01-PX01
   // Check_TON[52] : +ST020-CNV05-VM01-PX02
   // Check_TON[53] : +ST020-CNV05-VM01-PX03
   // Check_TON[54] : +ST020-CNV05-VM01-PX04
   // Check_TON[55] : +ST020-CNV05-VM01-PX05
   // Check_TON[56] : +ST020-CNV05-VM01-PX06
   // Check_TON[57] : +ST020-CNV05-VM01-PX07
   // Check_TON[58] : +ST020-CNV05-VM01-PX08
   // Check_TON[59] : +ST020-CNV05-VM01-PX09
   // Check_TON[60] : +ST020-CNV05-VM01-PX11
   // Check_TON[61] : +ST020-CNV05-VM01-PX10
   // Check_TON[62] : +ST020-CNV05-VM01-PX12
   // Check_TON[63] : +ST020-CNV05-VM01-PX13
   // Check_TON[64] : +ST020-CNV05-VM01-PX14
   // Check_TON[65] : +ST020-CNV05-VM01-PX15
   // Check_TON[66] : +ST020-CNV05-VM01-PX16
   // Check_TON[67] : +ST020-CNV05-VM01-PX17
   // Check_TON[68] : +ST020-CNV05-VM01-PX19
   // Check_TON[69] : +ST020-CNV05-VM01-PX20
   // Check_TON[70] : +ST020-CNV05-VM01-PX25
   // Check_TON[71] : +ST020-CNV05-VM01-PX21
   // Check_TON[72] : +ST020-CNV05-VM01-PX22
   // Check_TON[73] : +ST020-CNV05-VM01-PX23
   // Check_TON[74] : +ST020-CNV05-PX40
   // Check_TON[75] : +ST020-CNV05-PX41
   // Check_TON[76] : +ST020-CNV05-PX42
   // Check_TON[77] : +ST020-CNV05-PEY01
   // Check_TON[78] : +ST020-CNV05-PEY02
   // Check_TON[79] : +ST020-CNV05-PEY03
   // Check_TON[80] : +ST020-CNV05-PEY04
   // Check_TON[81] : +ST020-TL01-PX01
   // Check_TON[82] : +ST020-TL01-PX02
   // Check_TON[83] : +ST020-TL01-PX03
   // Check_TON[84] : +ST020-TL01-PX04
   // Check_TON[85] : +ST020-TL01-PX05
   // Check_TON[86] : +ST020-TL01-PX06
   // Check_TON[87] : +ST020-TL01-PX07
   // Check_TON[88] : +ST020-TL01-PX08
   // Check_TON[89] : +ST020-TL01-PX09
   // Check_TON[90] : +ST020-TL01-PX10
   // Check_TON[91] : +ST020-TO01-PEY01
   // Check_TON[92] : +ST020-TL09-SX01
   // Check_TON[93] : +ST020-TL09-SX02
   // Check_TON[94] : +ST020-TO02-PEY01
   // Check_TON[95] : +ST020-TL10-SX01
   // Check_TON[96] : +ST020-TL10-SX02
   // Check_TON[97] : +ST020-TO04-PEY01
   // Check_TON[98] : +ST020-TO04-PEY02
   // Check_TON[99] : +ST020-TL12-SX01
   // Check_TON[100] : +ST025-TL01- PX01
   // Check_TON[101] : +ST025-TL01- PX02
   // Check_TON[102] : +ST025-TL01- PX03
   // Check_TON[103] : +ST025-TL01- PX04
   // Check_TON[104] : +ST025-TL02- PX01
   // Check_TON[105] : +ST025-TL02- PX02
   // Check_TON[106] : +ST025-TL02- PX03
   // Check_TON[107] : +ST025-TL02- PX04
   // Check_TON[108] : +ST030-TL01- PX01
   // Check_TON[109] : +ST030-TL01- PX02
   // Check_TON[110] : +ST030-TL01- PX03
   // Check_TON[111] : +ST030-TL01- PX04
   // Check_TON[112] : +ST030-TL01- PX05
   // Check_TON[113] : +ST030-TL01- PX06
   // Check_TON[114] : +ST030-TL01- PX07
   // Check_TON[115] : +ST030-TL01- PX08
   // Check_TON[116] : +ST030-TL01- PX09
   // Check_TON[117] : +ST030-TL01- PX10
   // Check_TON[118] : +ST030-TL03- PX01
   // Check_TON[119] : +ST030-TL03- PX02
   // Check_TON[120] : +ST030-TL04- PX01
   // Check_TON[121] : +ST030-TL04- PX02
   // Check_TON[122] : +ST010-PX01
   // Check_TON[123] : +ST010-PX02
   // Check_TON[124] : +ST030-TL01- PX11
   // Check_TON[125] : +ST010-OffLine_PX01
   // Check_TON[126] : +ST010-OffLine_PX02
   // Check_TON[127] : ST020_LFT01_Repair
   // Check_TON[128] : ST030_LFT01_Repair
   // Check_TON[129] : ST035_LFT01_Repair
   // Check_TON[130] : +ST020-CNV0-PX39 TakeposBypass
   // Check_TON[131] : +ST030-TL03- PX03
   // Check_TON[132] : +ST030-TL03- PX04
   // Check_TON[133] : +ST030-TL04- PX03
   // Check_TON[134] : +ST030-TL04- PX04
END_DATA_BLOCK

DATA_BLOCK "GLOBAL_PROCESS_COMP_HMI_IF_DB"   // DB212
{ S7_Optimized_Access := 'TRUE' }
// stored: AutoNumber false, MemoryReserve 100
   VAR
      PROCESS_COMP { S7_SetPoint := 'True'} : Array[0..20] of "MISC_PROCESS_COMP_HMI_UDT";
   END_VAR
BEGIN
   // PROCESS_COMP[0] : +ST010-TL01
   // PROCESS_COMP[1] : +ST010-TL02
   // PROCESS_COMP[2] : +ST020-TL01
   // PROCESS_COMP[3] : +ST020-TL02
   // PROCESS_COMP[4] : +ST020-TL01
   // PROCESS_COMP[5] : +ST020-TL09
   // PROCESS_COMP[6] : +ST020-TL10
   // PROCESS_COMP[7] : +ST020-TL12
   // PROCESS_COMP[10] : +ST025-TL01
   // PROCESS_COMP[11] : +ST025-TL02
   // PROCESS_COMP[12] : +ST030-TL01
   // PROCESS_COMP[13] : +ST030-TL03
   // PROCESS_COMP[14] : +ST030-TL04
   // PROCESS_COMP[15] : +ST020-CNV04
   // PROCESS_COMP[16] : +ST020-CNV05
   // PROCESS_COMP[17] : +ST020-CNV06
END_DATA_BLOCK

DATA_BLOCK "GLOBAL_PROCESS_STOP_HMI_IF_DB"   // DB213
{ S7_Optimized_Access := 'TRUE' }
// stored: AutoNumber false, MemoryReserve 100
   VAR
      PROCESS_STOP { S7_SetPoint := 'True'} : Array[0..5] of "MISC_PROCESS_STOP_HMI_UDT";
   END_VAR
BEGIN
   // PROCESS_STOP[1] : +ST020-TL01
   // PROCESS_STOP[2] : +ST025-TL01
   // PROCESS_STOP[3] : +ST025-TL02
   // PROCESS_STOP[4] : +ST030-TL01
END_DATA_BLOCK

DATA_BLOCK "GLOBAL_ROBOT_DATA_DB"   // DB214
{ S7_Optimized_Access := 'TRUE' }
// stored: AutoNumber false, MemoryReserve 100
   VAR RETAIN
      Robot_HS_History_Data { ExternalWritable := 'False'} : Array[0..19] of "HS_HISTORY_EXTERNAL_UDT";
   END_VAR
BEGIN
END_DATA_BLOCK

DATA_BLOCK "GLOBAL_ROBOT_HMI_IF_DB"   // DB215
{ S7_Optimized_Access := 'TRUE' }
// stored: AutoNumber false, MemoryReserve 100
   VAR RETAIN
      Robot : Array[0..19] of "ROBOT_INTERFACE_HMI_UDT";
      Robot_HS { S7_SetPoint := 'True'} : Array[0..19] of "HS_HISTORY_HMI_UDT";
   END_VAR
BEGIN
   // Robot[1] : +ST020-RB01
   // Robot[2] : +ST020-RB02
   // Robot[3] : +ST020-RB03
   // Robot[4] : +ST020-RB04
   // Robot[5] : +ST020-RB06
   // Robot[6] : +ST025-RB01
   // Robot[7] : +ST025-RB02
   // Robot[8] : +ST030-RB01
   // Robot[9] : +ST030-RB02
   // Robot[10] : +ST030-RB03
   // Robot[11] : +ST030-RB04
END_DATA_BLOCK

DATA_BLOCK "GLOBAL_SERVICE_DB"   // DB218
{ S7_Optimized_Access := 'TRUE' }
// stored: AutoNumber false, MemoryReserve 100
   VAR RETAIN
      Service_Req : Array[0..10] of "ROBOT_GLOBAL_SRV_UDT";
   END_VAR
BEGIN
   // Service_Req[5] : OPMODE5
   // Service_Req[6] : OPMODE6
END_DATA_BLOCK

DATA_BLOCK "GLOBAL_Sensing_HMI_IF_DB"   // DB217
{ S7_Optimized_Access := 'TRUE' }
// stored: AutoNumber false, MemoryReserve 100
   VAR
      Sensing { S7_SetPoint := 'True'} : Array[0..1] of "KEYENCE_HMI_IF_UDT";
   END_VAR
BEGIN
END_DATA_BLOCK

DATA_BLOCK "GLOBAL_USER_ALARM_HMI_IF_DB"   // DB219
{ S7_Optimized_Access := 'TRUE' }
// stored: AutoNumber false, MemoryReserve 100
   VAR
      GLOBAL_USER_ALARM : Array[1..30] of "TEC_UNIT_HMI_UDT";
   END_VAR
BEGIN
END_DATA_BLOCK

DATA_BLOCK "GLOBAL_VALVE_HMI_IF_DB"   // DB220
{ S7_Optimized_Access := 'TRUE' }
// stored: AutoNumber false, MemoryReserve 100
   VAR RETAIN
      Valve { S7_SetPoint := 'True'} : Array[0..100] of "VALVE_HMI_UDT";
   END_VAR
BEGIN
   // Valve[1] : 左外上下缸
   // Valve[2] : 左外吸盘真空阀
END_DATA_BLOCK

DATA_BLOCK "1200_s7_1500"   // DB7
{ S7_Optimized_Access := 'FALSE' }
   VAR
      位1 : Bool;
      位2 : Bool;
      位3 : Bool;
      位4 : Bool;
      位5 : Bool;
      位6 : Bool;
      位7 : Bool;
      位8 : Bool;
      位9 : Bool;
      位10 : Bool;
      位11 : Bool;
      位12 : Bool;
      位13 : Bool;
      位14 : Bool;
      位15 : Bool;
      位16 : Bool;
      位17 : Bool;
      位18 : Bool;
      位19 : Bool;
      位20 : Bool;
      位21 : Bool;
      位22 : Bool;
      位23 : Bool;
      位24 : Bool;
      位25 : Bool;
      位26 : Bool;
      位27 : Bool;
      位28 : Bool;
      位29 : Bool;
      位30 : Bool;
      整型1 : Int;
      整型2 : Int;
      整型3 : Int;
      整型4 : Int;
      整型5 : Int;
      整型6 : Int;
      整型7 : Int;
      整型8 : Int;
      整型9 : Int;
      整型10 : Int;
      浮点数1 : Real;
      浮点数2 : Real;
      浮点数3 : Real;
      浮点数4 : Real;
      浮点数5 : Real;
      浮点数6 : Real;
      浮点数7 : Real;
      浮点数8 : Real;
      浮点数9 : Real;
      浮点数10 : Real;
      浮点数11 : Real;
      浮点数12 : Real;
      浮点数13 : Real;
      浮点数14 : Real;
      浮点数15 : Real;
      浮点数16 : Real;
      浮点数17 : Real;
      浮点数18 : Real;
      浮点数19 : Real;
   END_VAR
BEGIN
END_DATA_BLOCK

DATA_BLOCK "1500_s7_1200"   // DB6
{ S7_Optimized_Access := 'FALSE' }
   VAR
      位1 : Bool;
      位2 : Bool;
      位3 : Bool;
      位4 : Bool;
      位5 : Bool;
      位6 : Bool;
      位7 : Bool;
      位8 : Bool;
      位9 : Bool;
      位10 : Bool;
      位11 : Bool;
      位12 : Bool;
      位13 : Bool;
      位14 : Bool;
      位15 : Bool;
      位16 : Bool;
      位17 : Bool;
      位18 : Bool;
      位19 : Bool;
      位20 : Bool;
      位21 : Bool;
      位22 : Bool;
      位23 : Bool;
      位24 : Bool;
      位25 : Bool;
      位26 : Bool;
      位27 : Bool;
      位28 : Bool;
      位29 : Bool;
      位30 : Bool;
      整型1 : Int;
      整型2 : Int;
      整型3 : Int;
      整型4 : Int;
      整型5 : Int;
      整型6 : Int;
      整型7 : Int;
      整型8 : Int;
      整型9 : Int;
      整型10 : Int;
      浮点数1 : Real;
      浮点数2 : Real;
      浮点数3 : Real;
      浮点数4 : Real;
      浮点数5 : Real;
      浮点数6 : Real;
      浮点数7 : Real;
      浮点数8 : Real;
      浮点数9 : Real;
      浮点数10 : Real;
      浮点数11 : Real;
      浮点数12 : Real;
      浮点数13 : Real;
      浮点数14 : Real;
      浮点数15 : Real;
      浮点数16 : Real;
      浮点数17 : Real;
      浮点数18 : Real;
      浮点数19 : Real;
   END_VAR
BEGIN
END_DATA_BLOCK

DATA_BLOCK "1500_s7_G2"   // DB2
{ S7_Optimized_Access := 'FALSE' }
   VAR
      位1 : Bool;
      位2 : Bool;
      位3 : Bool;
      位4 : Bool;
      位5 : Bool;
      位6 : Bool;
      位7 : Bool;
      位8 : Bool;
      位9 : Bool;
      位10 : Bool;
      位11 : Bool;
      位12 : Bool;
      位13 : Bool;
      位14 : Bool;
      位15 : Bool;
      位16 : Bool;
      位17 : Bool;
      位18 : Bool;
      位19 : Bool;
      位20 : Bool;
      位21 : Bool;
      位22 : Bool;
      位23 : Bool;
      位24 : Bool;
      位25 : Bool;
      位26 : Bool;
      位27 : Bool;
      位28 : Bool;
      位29 : Bool;
      位30 : Bool;
      整型1 : Int;
      整型2 : Int;
      整型3 : Int;
      整型4 : Int;
      整型5 : Int;
      整型6 : Int;
      整型7 : Int;
      整型8 : Int;
      整型9 : Int;
      整型10 : Int;
      浮点数1 : Real;
      浮点数2 : Real;
      浮点数3 : Real;
      浮点数4 : Real;
      浮点数5 : Real;
      浮点数6 : Real;
      浮点数7 : Real;
      浮点数8 : Real;
      浮点数9 : Real;
      浮点数10 : Real;
      浮点数11 : Real;
      浮点数12 : Real;
      浮点数13 : Real;
      浮点数14 : Real;
      浮点数15 : Real;
      浮点数16 : Real;
      浮点数17 : Real;
      浮点数18 : Real;
      浮点数19 : Real;
   END_VAR
BEGIN
END_DATA_BLOCK

DATA_BLOCK "G2_s7_1500"   // DB4
{ S7_Optimized_Access := 'FALSE' }
   VAR
      位1 : Bool;
      位2 : Bool;
      位3 : Bool;
      位4 : Bool;
      位5 : Bool;
      位6 : Bool;
      位7 : Bool;
      位8 : Bool;
      位9 : Bool;
      位10 : Bool;
      位11 : Bool;
      位12 : Bool;
      位13 : Bool;
      位14 : Bool;
      位15 : Bool;
      位16 : Bool;
      位17 : Bool;
      位18 : Bool;
      位19 : Bool;
      位20 : Bool;
      位21 : Bool;
      位22 : Bool;
      位23 : Bool;
      位24 : Bool;
      位25 : Bool;
      位26 : Bool;
      位27 : Bool;
      位28 : Bool;
      位29 : Bool;
      位30 : Bool;
      整型1 : Int;
      整型2 : Int;
      整型3 : Int;
      整型4 : Int;
      整型5 : Int;
      整型6 : Int;
      整型7 : Int;
      整型8 : Int;
      整型9 : Int;
      整型10 : Int;
      浮点数1 : Real;
      浮点数2 : Real;
      浮点数3 : Real;
      浮点数4 : Real;
      浮点数5 : Real;
      浮点数6 : Real;
      浮点数7 : Real;
      浮点数8 : Real;
      浮点数9 : Real;
      浮点数10 : Real;
      浮点数11 : Real;
      浮点数12 : Real;
      浮点数13 : Real;
      浮点数14 : Real;
      浮点数15 : Real;
      浮点数16 : Real;
      浮点数17 : Real;
      浮点数18 : Real;
      浮点数19 : Real;
   END_VAR
BEGIN
END_DATA_BLOCK

DATA_BLOCK "HMI_AlarmData"   // DB20220
{ S7_Optimized_Access := 'TRUE' }
// stored: AutoNumber false, MemoryReserve 100
   VAR
      "Word" : Array[0..7] of Word;
   END_VAR
BEGIN
   // "Word"[0] : MES
END_DATA_BLOCK

